LIN {X 771.523, Y -384.331, Z 83.55, A 0, B 90, C -0, E1 0, E2 0, E3 0, E4 0} C_DIS
LIN {X 767.677, Y -378.417, Z 83.55, A 0, B 90, C -0, E1 0, E2 0, E3 0, E4 0} C_DIS
LIN {X 766.611, Y -377.585, Z 83.55, A 0, B 90, C -0, E1 0, E2 0, E3 0, E4 0} C_DIS
LIN {X 765.394, Y -378.227, Z 83.55, A 0, B 90, C -0, E1 0, E2 0, E3 0, E4 0} C_DIS
LIN {X 760.024, Y -382.801, Z 83.55, A 0, B 90, C -0, E1 0, E2 0, E3 0, E4 0} C_DIS
LIN {X 758.756, Y -383.361, Z 83.55, A 0, B 90, C -0, E1 0, E2 0, E3 0, E4 0} C_DIS
LIN {X 757.411, Y -383.004, Z 83.55, A 0, B 90, C -0, E1 0, E2 0, E3 0, E4 0} C_DIS
LIN {X 751.124, Y -379.806, Z 83.55, A 0, B 90, C -0, E1 0, E2 0, E3 0, E4 0} C_DIS
LIN {X 749.785, Y -379.619, Z 83.55, A 0, B 90, C -0, E1 0, E2 0, E3 0, E4 0} C_DIS
LIN {X 749.052, Y -380.783, Z 83.55, A 0, B 90, C -0, E1 0, E2 0, E3 0, E4 0} C_DIS
LIN {X 746.688, Y -387.429, Z 83.55, A 0, B 90, C -0, E1 0, E2 0, E3 0, E4 0} C_DIS
LIN {X 745.87, Y -388.548, Z 83.55, A 0, B 90, C -0, E1 0, E2 0, E3 0, E4 0} C_DIS
LIN {X 744.527, Y -388.912, Z 83.55, A 0, B 90, C -0, E1 0, E2 0, E3 0, E4 0} C_DIS
LIN {X 737.483, Y -389.285, Z 83.55, A 0, B 90, C -0, E1 0, E2 0, E3 0, E4 0} C_DIS
LIN {X 736.23, Y -389.793, Z 83.55, A 0, B 90, C -0, E1 0, E2 0, E3 0, E4 0} C_DIS
LIN {X 736.177, Y -391.167, Z 83.55, A 0, B 90, C -0, E1 0, E2 0, E3 0, E4 0} C_DIS
LIN {X 737.453, Y -398.105, Z 83.55, A 0, B 90, C -0, E1 0, E2 0, E3 0, E4 0} C_DIS
LIN {X 737.304, Y -399.483, Z 83.55, A 0, B 90, C -0, E1 0, E2 0, E3 0, E4 0} C_DIS
LIN {X 736.323, Y -400.469, Z 83.55, A 0, B 90, C -0, E1 0, E2 0, E3 0, E4 0} C_DIS
LIN {X 730.41, Y -404.315, Z 83.55, A 0, B 90, C -0, E1 0, E2 0, E3 0, E4 0} C_DIS
LIN {X 729.578, Y -405.381, Z 83.55, A 0, B 90, C -0, E1 0, E2 0, E3 0, E4 0} C_DIS
LIN {X 730.22, Y -406.598, Z 83.55, A 0, B 90, C -0, E1 0, E2 0, E3 0, E4 0} C_DIS
LIN {X 734.793, Y -411.969, Z 83.55, A 0, B 90, C -0, E1 0, E2 0, E3 0, E4 0} C_DIS
LIN {X 735.354, Y -413.236, Z 83.55, A 0, B 90, C -0, E1 0, E2 0, E3 0, E4 0} C_DIS
LIN {X 734.997, Y -414.581, Z 83.55, A 0, B 90, C -0, E1 0, E2 0, E3 0, E4 0} C_DIS
LIN {X 731.798, Y -420.868, Z 83.55, A 0, B 90, C -0, E1 0, E2 0, E3 0, E4 0} C_DIS
LIN {X 731.611, Y -422.208, Z 83.55, A 0, B 90, C -0, E1 0, E2 0, E3 0, E4 0} C_DIS
LIN {X 732.775, Y -422.94, Z 83.55, A 0, B 90, C -0, E1 0, E2 0, E3 0, E4 0} C_DIS
LIN {X 739.421, Y -425.305, Z 83.55, A 0, B 90, C -0, E1 0, E2 0, E3 0, E4 0} C_DIS
LIN {X 740.541, Y -426.122, Z 83.55, A 0, B 90, C -0, E1 0, E2 0, E3 0, E4 0} C_DIS
LIN {X 740.904, Y -427.465, Z 83.55, A 0, B 90, C -0, E1 0, E2 0, E3 0, E4 0} C_DIS
LIN {X 741.278, Y -434.509, Z 83.55, A 0, B 90, C -0, E1 0, E2 0, E3 0, E4 0} C_DIS
LIN {X 741.785, Y -435.763, Z 83.55, A 0, B 90, C -0, E1 0, E2 0, E3 0, E4 0} C_DIS
LIN {X 743.16, Y -435.815, Z 83.55, A 0, B 90, C -0, E1 0, E2 0, E3 0, E4 0} C_DIS
LIN {X 750.098, Y -434.54, Z 83.55, A 0, B 90, C -0, E1 0, E2 0, E3 0, E4 0} C_DIS
LIN {X 751.476, Y -434.688, Z 83.55, A 0, B 90, C -0, E1 0, E2 0, E3 0, E4 0} C_DIS
LIN {X 752.462, Y -435.669, Z 83.55, A 0, B 90, C -0, E1 0, E2 0, E3 0, E4 0} C_DIS
LIN {X 756.308, Y -441.583, Z 83.55, A 0, B 90, C -0, E1 0, E2 0, E3 0, E4 0} C_DIS
LIN {X 757.374, Y -442.415, Z 83.55, A 0, B 90, C -0, E1 0, E2 0, E3 0, E4 0} C_DIS
LIN {X 758.591, Y -441.773, Z 83.55, A 0, B 90, C -0, E1 0, E2 0, E3 0, E4 0} C_DIS
LIN {X 763.961, Y -437.199, Z 83.55, A 0, B 90, C -0, E1 0, E2 0, E3 0, E4 0} C_DIS
LIN {X 765.229, Y -436.639, Z 83.55, A 0, B 90, C -0, E1 0, E2 0, E3 0, E4 0} C_DIS
LIN {X 766.573, Y -436.996, Z 83.55, A 0, B 90, C -0, E1 0, E2 0, E3 0, E4 0} C_DIS
LIN {X 772.861, Y -440.194, Z 83.55, A 0, B 90, C -0, E1 0, E2 0, E3 0, E4 0} C_DIS
LIN {X 774.2, Y -440.381, Z 83.55, A 0, B 90, C -0, E1 0, E2 0, E3 0, E4 0} C_DIS
LIN {X 774.933, Y -439.217, Z 83.55, A 0, B 90, C -0, E1 0, E2 0, E3 0, E4 0} C_DIS
LIN {X 777.297, Y -432.571, Z 83.55, A 0, B 90, C -0, E1 0, E2 0, E3 0, E4 0} C_DIS
LIN {X 778.115, Y -431.452, Z 83.55, A 0, B 90, C -0, E1 0, E2 0, E3 0, E4 0} C_DIS
LIN {X 779.458, Y -431.088, Z 83.55, A 0, B 90, C -0, E1 0, E2 0, E3 0, E4 0} C_DIS
LIN {X 786.502, Y -430.715, Z 83.55, A 0, B 90, C -0, E1 0, E2 0, E3 0, E4 0} C_DIS
LIN {X 787.755, Y -430.207, Z 83.55, A 0, B 90, C -0, E1 0, E2 0, E3 0, E4 0} C_DIS
LIN {X 787.808, Y -428.833, Z 83.55, A 0, B 90, C -0, E1 0, E2 0, E3 0, E4 0} C_DIS
LIN {X 786.532, Y -421.895, Z 83.55, A 0, B 90, C -0, E1 0, E2 0, E3 0, E4 0} C_DIS
LIN {X 786.681, Y -420.517, Z 83.55, A 0, B 90, C -0, E1 0, E2 0, E3 0, E4 0} C_DIS
LIN {X 787.662, Y -419.531, Z 83.55, A 0, B 90, C -0, E1 0, E2 0, E3 0, E4 0} C_DIS
LIN {X 793.575, Y -415.685, Z 83.55, A 0, B 90, C -0, E1 0, E2 0, E3 0, E4 0} C_DIS
LIN {X 794.407, Y -414.619, Z 83.55, A 0, B 90, C -0, E1 0, E2 0, E3 0, E4 0} C_DIS
LIN {X 793.765, Y -413.402, Z 83.55, A 0, B 90, C -0, E1 0, E2 0, E3 0, E4 0} C_DIS
LIN {X 789.192, Y -408.031, Z 83.55, A 0, B 90, C -0, E1 0, E2 0, E3 0, E4 0} C_DIS
LIN {X 788.631, Y -406.764, Z 83.55, A 0, B 90, C -0, E1 0, E2 0, E3 0, E4 0} C_DIS
LIN {X 788.988, Y -405.419, Z 83.55, A 0, B 90, C -0, E1 0, E2 0, E3 0, E4 0} C_DIS
LIN {X 792.186, Y -399.132, Z 83.55, A 0, B 90, C -0, E1 0, E2 0, E3 0, E4 0} C_DIS
LIN {X 792.374, Y -397.792, Z 83.55, A 0, B 90, C -0, E1 0, E2 0, E3 0, E4 0} C_DIS
LIN {X 791.209, Y -397.06, Z 83.55, A 0, B 90, C -0, E1 0, E2 0, E3 0, E4 0} C_DIS
LIN {X 784.564, Y -394.695, Z 83.55, A 0, B 90, C -0, E1 0, E2 0, E3 0, E4 0} C_DIS
LIN {X 783.444, Y -393.878, Z 83.55, A 0, B 90, C -0, E1 0, E2 0, E3 0, E4 0} C_DIS
LIN {X 783.081, Y -392.535, Z 83.55, A 0, B 90, C -0, E1 0, E2 0, E3 0, E4 0} C_DIS
LIN {X 782.707, Y -385.491, Z 83.55, A 0, B 90, C -0, E1 0, E2 0, E3 0, E4 0} C_DIS
LIN {X 782.2, Y -384.237, Z 83.55, A 0, B 90, C -0, E1 0, E2 0, E3 0, E4 0} C_DIS
LIN {X 780.825, Y -384.185, Z 83.55, A 0, B 90, C -0, E1 0, E2 0, E3 0, E4 0} C_DIS
LIN {X 775.275, Y -385.205, Z 83.55, A 0, B 90, C -0, E1 0, E2 0, E3 0, E4 0} C_DIS
LIN {X 773.608, Y -385.498, Z 84.2, A 0, B 90, C -0, E1 0, E2 0, E3 0, E4 0} C_DIS
LIN {X 772.237, Y -385.362, Z 84.2, A 0, B 90, C -0, E1 0, E2 0, E3 0, E4 0} C_DIS
LIN {X 771.248, Y -384.395, Z 84.2, A 0, B 90, C -0, E1 0, E2 0, E3 0, E4 0} C_DIS
LIN {X 767.373, Y -378.549, Z 84.2, A 0, B 90, C -0, E1 0, E2 0, E3 0, E4 0} C_DIS
LIN {X 766.306, Y -377.731, Z 84.2, A 0, B 90, C -0, E1 0, E2 0, E3 0, E4 0} C_DIS
LIN {X 765.101, Y -378.379, Z 84.2, A 0, B 90, C -0, E1 0, E2 0, E3 0, E4 0} C_DIS
LIN {X 759.801, Y -382.973, Z 84.2, A 0, B 90, C -0, E1 0, E2 0, E3 0, E4 0} C_DIS
LIN {X 758.545, Y -383.541, Z 84.2, A 0, B 90, C -0, E1 0, E2 0, E3 0, E4 0} C_DIS
LIN {X 757.205, Y -383.198, Z 84.2, A 0, B 90, C -0, E1 0, E2 0, E3 0, E4 0} C_DIS
LIN {X 750.926, Y -380.072, Z 84.2, A 0, B 90, C -0, E1 0, E2 0, E3 0, E4 0} C_DIS
LIN {X 749.593, Y -379.897, Z 84.2, A 0, B 90, C -0, E1 0, E2 0, E3 0, E4 0} C_DIS
LIN {X 748.875, Y -381.061, Z 84.2, A 0, B 90, C -0, E1 0, E2 0, E3 0, E4 0} C_DIS
LIN {X 746.581, Y -387.69, Z 84.2, A 0, B 90, C -0, E1 0, E2 0, E3 0, E4 0} C_DIS
LIN {X 745.778, Y -388.81, Z 84.2, A 0, B 90, C -0, E1 0, E2 0, E3 0, E4 0} C_DIS
LIN {X 744.446, Y -389.182, Z 84.2, A 0, B 90, C -0, E1 0, E2 0, E3 0, E4 0} C_DIS
LIN {X 737.445, Y -389.615, Z 84.2, A 0, B 90, C -0, E1 0, E2 0, E3 0, E4 0} C_DIS
LIN {X 736.203, Y -390.13, Z 84.2, A 0, B 90, C -0, E1 0, E2 0, E3 0, E4 0} C_DIS
LIN {X 736.163, Y -391.497, Z 84.2, A 0, B 90, C -0, E1 0, E2 0, E3 0, E4 0} C_DIS
LIN {X 737.491, Y -398.384, Z 84.2, A 0, B 90, C -0, E1 0, E2 0, E3 0, E4 0} C_DIS
LIN {X 737.355, Y -399.756, Z 84.2, A 0, B 90, C -0, E1 0, E2 0, E3 0, E4 0} C_DIS
LIN {X 736.388, Y -400.745, Z 84.2, A 0, B 90, C -0, E1 0, E2 0, E3 0, E4 0} C_DIS
LIN {X 730.541, Y -404.619, Z 84.2, A 0, B 90, C -0, E1 0, E2 0, E3 0, E4 0} C_DIS
LIN {X 729.723, Y -405.687, Z 84.2, A 0, B 90, C -0, E1 0, E2 0, E3 0, E4 0} C_DIS
LIN {X 730.372, Y -406.891, Z 84.2, A 0, B 90, C -0, E1 0, E2 0, E3 0, E4 0} C_DIS
LIN {X 734.965, Y -412.191, Z 84.2, A 0, B 90, C -0, E1 0, E2 0, E3 0, E4 0} C_DIS
LIN {X 735.534, Y -413.447, Z 84.2, A 0, B 90, C -0, E1 0, E2 0, E3 0, E4 0} C_DIS
LIN {X 735.19, Y -414.787, Z 84.2, A 0, B 90, C -0, E1 0, E2 0, E3 0, E4 0} C_DIS
LIN {X 732.064, Y -421.066, Z 84.2, A 0, B 90, C -0, E1 0, E2 0, E3 0, E4 0} C_DIS
LIN {X 731.89, Y -422.399, Z 84.2, A 0, B 90, C -0, E1 0, E2 0, E3 0, E4 0} C_DIS
LIN {X 733.054, Y -423.118, Z 84.2, A 0, B 90, C -0, E1 0, E2 0, E3 0, E4 0} C_DIS
LIN {X 739.682, Y -425.411, Z 84.2, A 0, B 90, C -0, E1 0, E2 0, E3 0, E4 0} C_DIS
LIN {X 740.802, Y -426.215, Z 84.2, A 0, B 90, C -0, E1 0, E2 0, E3 0, E4 0} C_DIS
LIN {X 741.175, Y -427.547, Z 84.2, A 0, B 90, C -0, E1 0, E2 0, E3 0, E4 0} C_DIS
LIN {X 741.607, Y -434.547, Z 84.2, A 0, B 90, C -0, E1 0, E2 0, E3 0, E4 0} C_DIS
LIN {X 742.122, Y -435.79, Z 84.2, A 0, B 90, C -0, E1 0, E2 0, E3 0, E4 0} C_DIS
LIN {X 743.49, Y -435.83, Z 84.2, A 0, B 90, C -0, E1 0, E2 0, E3 0, E4 0} C_DIS
LIN {X 750.377, Y -434.502, Z 84.2, A 0, B 90, C -0, E1 0, E2 0, E3 0, E4 0} C_DIS
LIN {X 751.748, Y -434.638, Z 84.2, A 0, B 90, C -0, E1 0, E2 0, E3 0, E4 0} C_DIS
LIN {X 752.737, Y -435.605, Z 84.2, A 0, B 90, C -0, E1 0, E2 0, E3 0, E4 0} C_DIS
LIN {X 756.612, Y -441.451, Z 84.2, A 0, B 90, C -0, E1 0, E2 0, E3 0, E4 0} C_DIS
LIN {X 757.679, Y -442.269, Z 84.2, A 0, B 90, C -0, E1 0, E2 0, E3 0, E4 0} C_DIS
LIN {X 758.884, Y -441.621, Z 84.2, A 0, B 90, C -0, E1 0, E2 0, E3 0, E4 0} C_DIS
LIN {X 764.184, Y -437.027, Z 84.2, A 0, B 90, C -0, E1 0, E2 0, E3 0, E4 0} C_DIS
LIN {X 765.44, Y -436.459, Z 84.2, A 0, B 90, C -0, E1 0, E2 0, E3 0, E4 0} C_DIS
LIN {X 766.78, Y -436.802, Z 84.2, A 0, B 90, C -0, E1 0, E2 0, E3 0, E4 0} C_DIS
LIN {X 773.058, Y -439.928, Z 84.2, A 0, B 90, C -0, E1 0, E2 0, E3 0, E4 0} C_DIS
LIN {X 774.392, Y -440.103, Z 84.2, A 0, B 90, C -0, E1 0, E2 0, E3 0, E4 0} C_DIS
LIN {X 775.11, Y -438.939, Z 84.2, A 0, B 90, C -0, E1 0, E2 0, E3 0, E4 0} C_DIS
LIN {X 777.404, Y -432.31, Z 84.2, A 0, B 90, C -0, E1 0, E2 0, E3 0, E4 0} C_DIS
LIN {X 778.207, Y -431.19, Z 84.2, A 0, B 90, C -0, E1 0, E2 0, E3 0, E4 0} C_DIS
LIN {X 779.539, Y -430.818, Z 84.2, A 0, B 90, C -0, E1 0, E2 0, E3 0, E4 0} C_DIS
LIN {X 786.54, Y -430.385, Z 84.2, A 0, B 90, C -0, E1 0, E2 0, E3 0, E4 0} C_DIS
LIN {X 787.782, Y -429.87, Z 84.2, A 0, B 90, C -0, E1 0, E2 0, E3 0, E4 0} C_DIS
LIN {X 787.822, Y -428.503, Z 84.2, A 0, B 90, C -0, E1 0, E2 0, E3 0, E4 0} C_DIS
LIN {X 786.494, Y -421.616, Z 84.2, A 0, B 90, C -0, E1 0, E2 0, E3 0, E4 0} C_DIS
LIN {X 786.63, Y -420.244, Z 84.2, A 0, B 90, C -0, E1 0, E2 0, E3 0, E4 0} C_DIS
LIN {X 787.597, Y -419.255, Z 84.2, A 0, B 90, C -0, E1 0, E2 0, E3 0, E4 0} C_DIS
LIN {X 793.444, Y -415.381, Z 84.2, A 0, B 90, C -0, E1 0, E2 0, E3 0, E4 0} C_DIS
LIN {X 794.262, Y -414.313, Z 84.2, A 0, B 90, C -0, E1 0, E2 0, E3 0, E4 0} C_DIS
LIN {X 793.613, Y -413.109, Z 84.2, A 0, B 90, C -0, E1 0, E2 0, E3 0, E4 0} C_DIS
LIN {X 789.02, Y -407.809, Z 84.2, A 0, B 90, C -0, E1 0, E2 0, E3 0, E4 0} C_DIS
LIN {X 788.451, Y -406.553, Z 84.2, A 0, B 90, C -0, E1 0, E2 0, E3 0, E4 0} C_DIS
LIN {X 788.795, Y -405.213, Z 84.2, A 0, B 90, C -0, E1 0, E2 0, E3 0, E4 0} C_DIS
LIN {X 791.92, Y -398.934, Z 84.2, A 0, B 90, C -0, E1 0, E2 0, E3 0, E4 0} C_DIS
LIN {X 792.095, Y -397.601, Z 84.2, A 0, B 90, C -0, E1 0, E2 0, E3 0, E4 0} C_DIS
LIN {X 790.931, Y -396.882, Z 84.2, A 0, B 90, C -0, E1 0, E2 0, E3 0, E4 0} C_DIS
LIN {X 784.303, Y -394.589, Z 84.2, A 0, B 90, C -0, E1 0, E2 0, E3 0, E4 0} C_DIS
LIN {X 783.183, Y -393.785, Z 84.2, A 0, B 90, C -0, E1 0, E2 0, E3 0, E4 0} C_DIS
LIN {X 782.81, Y -392.453, Z 84.2, A 0, B 90, C -0, E1 0, E2 0, E3 0, E4 0} C_DIS
LIN {X 782.378, Y -385.453, Z 84.2, A 0, B 90, C -0, E1 0, E2 0, E3 0, E4 0} C_DIS
LIN {X 781.862, Y -384.21, Z 84.2, A 0, B 90, C -0, E1 0, E2 0, E3 0, E4 0} C_DIS
LIN {X 780.495, Y -384.17, Z 84.2, A 0, B 90, C -0, E1 0, E2 0, E3 0, E4 0} C_DIS
LIN {X 774.986, Y -385.233, Z 84.2, A 0, B 90, C -0, E1 0, E2 0, E3 0, E4 0} C_DIS
LIN {X 773.332, Y -385.538, Z 84.85, A 0, B 90, C -0, E1 0, E2 0, E3 0, E4 0} C_DIS
LIN {X 771.966, Y -385.414, Z 84.85, A 0, B 90, C -0, E1 0, E2 0, E3 0, E4 0} C_DIS
LIN {X 770.975, Y -384.461, Z 84.85, A 0, B 90, C -0, E1 0, E2 0, E3 0, E4 0} C_DIS
LIN {X 767.072, Y -378.681, Z 84.85, A 0, B 90, C -0, E1 0, E2 0, E3 0, E4 0} C_DIS
LIN {X 766.004, Y -377.877, Z 84.85, A 0, B 90, C -0, E1 0, E2 0, E3 0, E4 0} C_DIS
LIN {X 764.812, Y -378.533, Z 84.85, A 0, B 90, C -0, E1 0, E2 0, E3 0, E4 0} C_DIS
LIN {X 759.581, Y -383.145, Z 84.85, A 0, B 90, C -0, E1 0, E2 0, E3 0, E4 0} C_DIS
LIN {X 758.337, Y -383.721, Z 84.85, A 0, B 90, C -0, E1 0, E2 0, E3 0, E4 0} C_DIS
LIN {X 757.002, Y -383.392, Z 84.85, A 0, B 90, C -0, E1 0, E2 0, E3 0, E4 0} C_DIS
LIN {X 750.732, Y -380.337, Z 84.85, A 0, B 90, C -0, E1 0, E2 0, E3 0, E4 0} C_DIS
LIN {X 749.405, Y -380.175, Z 84.85, A 0, B 90, C -0, E1 0, E2 0, E3 0, E4 0} C_DIS
LIN {X 748.701, Y -381.339, Z 84.85, A 0, B 90, C -0, E1 0, E2 0, E3 0, E4 0} C_DIS
LIN {X 746.477, Y -387.949, Z 84.85, A 0, B 90, C -0, E1 0, E2 0, E3 0, E4 0} C_DIS
LIN {X 745.688, Y -389.069, Z 84.85, A 0, B 90, C -0, E1 0, E2 0, E3 0, E4 0} C_DIS
LIN {X 744.367, Y -389.452, Z 84.85, A 0, B 90, C -0, E1 0, E2 0, E3 0, E4 0} C_DIS
LIN {X 737.409, Y -389.942, Z 84.85, A 0, B 90, C -0, E1 0, E2 0, E3 0, E4 0} C_DIS
LIN {X 736.179, Y -390.465, Z 84.85, A 0, B 90, C -0, E1 0, E2 0, E3 0, E4 0} C_DIS
LIN {X 736.151, Y -391.824, Z 84.85, A 0, B 90, C -0, E1 0, E2 0, E3 0, E4 0} C_DIS
LIN {X 737.53, Y -398.661, Z 84.85, A 0, B 90, C -0, E1 0, E2 0, E3 0, E4 0} C_DIS
LIN {X 737.407, Y -400.026, Z 84.85, A 0, B 90, C -0, E1 0, E2 0, E3 0, E4 0} C_DIS
LIN {X 736.454, Y -401.017, Z 84.85, A 0, B 90, C -0, E1 0, E2 0, E3 0, E4 0} C_DIS
LIN {X 730.674, Y -404.92, Z 84.85, A 0, B 90, C -0, E1 0, E2 0, E3 0, E4 0} C_DIS
LIN {X 729.87, Y -405.989, Z 84.85, A 0, B 90, C -0, E1 0, E2 0, E3 0, E4 0} C_DIS
LIN {X 730.525, Y -407.181, Z 84.85, A 0, B 90, C -0, E1 0, E2 0, E3 0, E4 0} C_DIS
LIN {X 735.138, Y -412.411, Z 84.85, A 0, B 90, C -0, E1 0, E2 0, E3 0, E4 0} C_DIS
LIN {X 735.714, Y -413.655, Z 84.85, A 0, B 90, C -0, E1 0, E2 0, E3 0, E4 0} C_DIS
LIN {X 735.384, Y -414.99, Z 84.85, A 0, B 90, C -0, E1 0, E2 0, E3 0, E4 0} C_DIS
LIN {X 732.33, Y -421.26, Z 84.85, A 0, B 90, C -0, E1 0, E2 0, E3 0, E4 0} C_DIS
LIN {X 732.168, Y -422.588, Z 84.85, A 0, B 90, C -0, E1 0, E2 0, E3 0, E4 0} C_DIS
LIN {X 733.331, Y -423.292, Z 84.85, A 0, B 90, C -0, E1 0, E2 0, E3 0, E4 0} C_DIS
LIN {X 739.941, Y -425.515, Z 84.85, A 0, B 90, C -0, E1 0, E2 0, E3 0, E4 0} C_DIS
LIN {X 741.062, Y -426.305, Z 84.85, A 0, B 90, C -0, E1 0, E2 0, E3 0, E4 0} C_DIS
LIN {X 741.444, Y -427.626, Z 84.85, A 0, B 90, C -0, E1 0, E2 0, E3 0, E4 0} C_DIS
LIN {X 741.934, Y -434.583, Z 84.85, A 0, B 90, C -0, E1 0, E2 0, E3 0, E4 0} C_DIS
LIN {X 742.457, Y -435.814, Z 84.85, A 0, B 90, C -0, E1 0, E2 0, E3 0, E4 0} C_DIS
LIN {X 743.817, Y -435.842, Z 84.85, A 0, B 90, C -0, E1 0, E2 0, E3 0, E4 0} C_DIS
LIN {X 750.653, Y -434.462, Z 84.85, A 0, B 90, C -0, E1 0, E2 0, E3 0, E4 0} C_DIS
LIN {X 752.018, Y -434.586, Z 84.85, A 0, B 90, C -0, E1 0, E2 0, E3 0, E4 0} C_DIS
LIN {X 753.01, Y -435.539, Z 84.85, A 0, B 90, C -0, E1 0, E2 0, E3 0, E4 0} C_DIS
LIN {X 756.913, Y -441.319, Z 84.85, A 0, B 90, C -0, E1 0, E2 0, E3 0, E4 0} C_DIS
LIN {X 757.981, Y -442.123, Z 84.85, A 0, B 90, C -0, E1 0, E2 0, E3 0, E4 0} C_DIS
LIN {X 759.173, Y -441.467, Z 84.85, A 0, B 90, C -0, E1 0, E2 0, E3 0, E4 0} C_DIS
LIN {X 764.404, Y -436.855, Z 84.85, A 0, B 90, C -0, E1 0, E2 0, E3 0, E4 0} C_DIS
LIN {X 765.648, Y -436.279, Z 84.85, A 0, B 90, C -0, E1 0, E2 0, E3 0, E4 0} C_DIS
LIN {X 766.983, Y -436.608, Z 84.85, A 0, B 90, C -0, E1 0, E2 0, E3 0, E4 0} C_DIS
LIN {X 773.253, Y -439.663, Z 84.85, A 0, B 90, C -0, E1 0, E2 0, E3 0, E4 0} C_DIS
LIN {X 774.58, Y -439.825, Z 84.85, A 0, B 90, C -0, E1 0, E2 0, E3 0, E4 0} C_DIS
LIN {X 775.284, Y -438.661, Z 84.85, A 0, B 90, C -0, E1 0, E2 0, E3 0, E4 0} C_DIS
LIN {X 777.508, Y -432.051, Z 84.85, A 0, B 90, C -0, E1 0, E2 0, E3 0, E4 0} C_DIS
LIN {X 778.297, Y -430.931, Z 84.85, A 0, B 90, C -0, E1 0, E2 0, E3 0, E4 0} C_DIS
LIN {X 779.618, Y -430.548, Z 84.85, A 0, B 90, C -0, E1 0, E2 0, E3 0, E4 0} C_DIS
LIN {X 786.576, Y -430.058, Z 84.85, A 0, B 90, C -0, E1 0, E2 0, E3 0, E4 0} C_DIS
LIN {X 787.806, Y -429.535, Z 84.85, A 0, B 90, C -0, E1 0, E2 0, E3 0, E4 0} C_DIS
LIN {X 787.834, Y -428.176, Z 84.85, A 0, B 90, C -0, E1 0, E2 0, E3 0, E4 0} C_DIS
LIN {X 786.455, Y -421.339, Z 84.85, A 0, B 90, C -0, E1 0, E2 0, E3 0, E4 0} C_DIS
LIN {X 786.578, Y -419.974, Z 84.85, A 0, B 90, C -0, E1 0, E2 0, E3 0, E4 0} C_DIS
LIN {X 787.531, Y -418.983, Z 84.85, A 0, B 90, C -0, E1 0, E2 0, E3 0, E4 0} C_DIS
LIN {X 793.311, Y -415.08, Z 84.85, A 0, B 90, C -0, E1 0, E2 0, E3 0, E4 0} C_DIS
LIN {X 794.115, Y -414.011, Z 84.85, A 0, B 90, C -0, E1 0, E2 0, E3 0, E4 0} C_DIS
LIN {X 793.46, Y -412.819, Z 84.85, A 0, B 90, C -0, E1 0, E2 0, E3 0, E4 0} C_DIS
LIN {X 788.847, Y -407.589, Z 84.85, A 0, B 90, C -0, E1 0, E2 0, E3 0, E4 0} C_DIS
LIN {X 788.271, Y -406.345, Z 84.85, A 0, B 90, C -0, E1 0, E2 0, E3 0, E4 0} C_DIS
LIN {X 788.601, Y -405.01, Z 84.85, A 0, B 90, C -0, E1 0, E2 0, E3 0, E4 0} C_DIS
LIN {X 791.655, Y -398.74, Z 84.85, A 0, B 90, C -0, E1 0, E2 0, E3 0, E4 0} C_DIS
LIN {X 791.817, Y -397.412, Z 84.85, A 0, B 90, C -0, E1 0, E2 0, E3 0, E4 0} C_DIS
LIN {X 790.654, Y -396.708, Z 84.85, A 0, B 90, C -0, E1 0, E2 0, E3 0, E4 0} C_DIS
LIN {X 784.044, Y -394.485, Z 84.85, A 0, B 90, C -0, E1 0, E2 0, E3 0, E4 0} C_DIS
LIN {X 782.923, Y -393.695, Z 84.85, A 0, B 90, C -0, E1 0, E2 0, E3 0, E4 0} C_DIS
LIN {X 782.541, Y -392.374, Z 84.85, A 0, B 90, C -0, E1 0, E2 0, E3 0, E4 0} C_DIS
LIN {X 782.051, Y -385.417, Z 84.85, A 0, B 90, C -0, E1 0, E2 0, E3 0, E4 0} C_DIS
LIN {X 781.528, Y -384.186, Z 84.85, A 0, B 90, C -0, E1 0, E2 0, E3 0, E4 0} C_DIS
LIN {X 780.168, Y -384.158, Z 84.85, A 0, B 90, C -0, E1 0, E2 0, E3 0, E4 0} C_DIS
LIN {X 774.699, Y -385.262, Z 84.85, A 0, B 90, C -0, E1 0, E2 0, E3 0, E4 0} C_DIS
LIN {X 773.057, Y -385.579, Z 85.5, A 0, B 90, C -0, E1 0, E2 0, E3 0, E4 0} C_DIS
LIN {X 771.699, Y -385.468, Z 85.5, A 0, B 90, C -0, E1 0, E2 0, E3 0, E4 0} C_DIS
LIN {X 770.705, Y -384.529, Z 85.5, A 0, B 90, C -0, E1 0, E2 0, E3 0, E4 0} C_DIS
LIN {X 766.775, Y -378.815, Z 85.5, A 0, B 90, C -0, E1 0, E2 0, E3 0, E4 0} C_DIS
LIN {X 765.706, Y -378.025, Z 85.5, A 0, B 90, C -0, E1 0, E2 0, E3 0, E4 0} C_DIS
LIN {X 764.526, Y -378.686, Z 85.5, A 0, B 90, C -0, E1 0, E2 0, E3 0, E4 0} C_DIS
LIN {X 759.364, Y -383.318, Z 85.5, A 0, B 90, C -0, E1 0, E2 0, E3 0, E4 0} C_DIS
LIN {X 758.133, Y -383.901, Z 85.5, A 0, B 90, C -0, E1 0, E2 0, E3 0, E4 0} C_DIS
LIN {X 756.802, Y -383.585, Z 85.5, A 0, B 90, C -0, E1 0, E2 0, E3 0, E4 0} C_DIS
LIN {X 750.541, Y -380.602, Z 85.5, A 0, B 90, C -0, E1 0, E2 0, E3 0, E4 0} C_DIS
LIN {X 749.22, Y -380.452, Z 85.5, A 0, B 90, C -0, E1 0, E2 0, E3 0, E4 0} C_DIS
LIN {X 748.53, Y -381.615, Z 85.5, A 0, B 90, C -0, E1 0, E2 0, E3 0, E4 0} C_DIS
LIN {X 746.376, Y -388.207, Z 85.5, A 0, B 90, C -0, E1 0, E2 0, E3 0, E4 0} C_DIS
LIN {X 745.6, Y -389.328, Z 85.5, A 0, B 90, C -0, E1 0, E2 0, E3 0, E4 0} C_DIS
LIN {X 744.29, Y -389.719, Z 85.5, A 0, B 90, C -0, E1 0, E2 0, E3 0, E4 0} C_DIS
LIN {X 737.377, Y -390.266, Z 85.5, A 0, B 90, C -0, E1 0, E2 0, E3 0, E4 0} C_DIS
LIN {X 736.157, Y -390.797, Z 85.5, A 0, B 90, C -0, E1 0, E2 0, E3 0, E4 0} C_DIS
LIN {X 736.141, Y -392.149, Z 85.5, A 0, B 90, C -0, E1 0, E2 0, E3 0, E4 0} C_DIS
LIN {X 737.571, Y -398.935, Z 85.5, A 0, B 90, C -0, E1 0, E2 0, E3 0, E4 0} C_DIS
LIN {X 737.46, Y -400.293, Z 85.5, A 0, B 90, C -0, E1 0, E2 0, E3 0, E4 0} C_DIS
LIN {X 736.521, Y -401.287, Z 85.5, A 0, B 90, C -0, E1 0, E2 0, E3 0, E4 0} C_DIS
LIN {X 730.807, Y -405.218, Z 85.5, A 0, B 90, C -0, E1 0, E2 0, E3 0, E4 0} C_DIS
LIN {X 730.017, Y -406.287, Z 85.5, A 0, B 90, C -0, E1 0, E2 0, E3 0, E4 0} C_DIS
LIN {X 730.679, Y -407.466, Z 85.5, A 0, B 90, C -0, E1 0, E2 0, E3 0, E4 0} C_DIS
LIN {X 735.311, Y -412.628, Z 85.5, A 0, B 90, C -0, E1 0, E2 0, E3 0, E4 0} C_DIS
LIN {X 735.894, Y -413.86, Z 85.5, A 0, B 90, C -0, E1 0, E2 0, E3 0, E4 0} C_DIS
LIN {X 735.577, Y -415.19, Z 85.5, A 0, B 90, C -0, E1 0, E2 0, E3 0, E4 0} C_DIS
LIN {X 732.594, Y -421.451, Z 85.5, A 0, B 90, C -0, E1 0, E2 0, E3 0, E4 0} C_DIS
LIN {X 732.444, Y -422.772, Z 85.5, A 0, B 90, C -0, E1 0, E2 0, E3 0, E4 0} C_DIS
LIN {X 733.607, Y -423.463, Z 85.5, A 0, B 90, C -0, E1 0, E2 0, E3 0, E4 0} C_DIS
LIN {X 740.199, Y -425.617, Z 85.5, A 0, B 90, C -0, E1 0, E2 0, E3 0, E4 0} C_DIS
LIN {X 741.32, Y -426.392, Z 85.5, A 0, B 90, C -0, E1 0, E2 0, E3 0, E4 0} C_DIS
LIN {X 741.712, Y -427.702, Z 85.5, A 0, B 90, C -0, E1 0, E2 0, E3 0, E4 0} C_DIS
LIN {X 742.258, Y -434.616, Z 85.5, A 0, B 90, C -0, E1 0, E2 0, E3 0, E4 0} C_DIS
LIN {X 742.789, Y -435.835, Z 85.5, A 0, B 90, C -0, E1 0, E2 0, E3 0, E4 0} C_DIS
LIN {X 744.142, Y -435.852, Z 85.5, A 0, B 90, C -0, E1 0, E2 0, E3 0, E4 0} C_DIS
LIN {X 750.927, Y -434.421, Z 85.5, A 0, B 90, C -0, E1 0, E2 0, E3 0, E4 0} C_DIS
LIN {X 752.286, Y -434.532, Z 85.5, A 0, B 90, C -0, E1 0, E2 0, E3 0, E4 0} C_DIS
LIN {X 753.28, Y -435.471, Z 85.5, A 0, B 90, C -0, E1 0, E2 0, E3 0, E4 0} C_DIS
LIN {X 757.21, Y -441.185, Z 85.5, A 0, B 90, C -0, E1 0, E2 0, E3 0, E4 0} C_DIS
LIN {X 758.279, Y -441.975, Z 85.5, A 0, B 90, C -0, E1 0, E2 0, E3 0, E4 0} C_DIS
LIN {X 759.459, Y -441.314, Z 85.5, A 0, B 90, C -0, E1 0, E2 0, E3 0, E4 0} C_DIS
LIN {X 764.62, Y -436.682, Z 85.5, A 0, B 90, C -0, E1 0, E2 0, E3 0, E4 0} C_DIS
LIN {X 765.852, Y -436.099, Z 85.5, A 0, B 90, C -0, E1 0, E2 0, E3 0, E4 0} C_DIS
LIN {X 767.183, Y -436.415, Z 85.5, A 0, B 90, C -0, E1 0, E2 0, E3 0, E4 0} C_DIS
LIN {X 773.443, Y -439.398, Z 85.5, A 0, B 90, C -0, E1 0, E2 0, E3 0, E4 0} C_DIS
LIN {X 774.765, Y -439.548, Z 85.5, A 0, B 90, C -0, E1 0, E2 0, E3 0, E4 0} C_DIS
LIN {X 775.455, Y -438.385, Z 85.5, A 0, B 90, C -0, E1 0, E2 0, E3 0, E4 0} C_DIS
LIN {X 777.609, Y -431.793, Z 85.5, A 0, B 90, C -0, E1 0, E2 0, E3 0, E4 0} C_DIS
LIN {X 778.385, Y -430.672, Z 85.5, A 0, B 90, C -0, E1 0, E2 0, E3 0, E4 0} C_DIS
LIN {X 779.695, Y -430.281, Z 85.5, A 0, B 90, C -0, E1 0, E2 0, E3 0, E4 0} C_DIS
LIN {X 786.608, Y -429.734, Z 85.5, A 0, B 90, C -0, E1 0, E2 0, E3 0, E4 0} C_DIS
LIN {X 787.828, Y -429.203, Z 85.5, A 0, B 90, C -0, E1 0, E2 0, E3 0, E4 0} C_DIS
LIN {X 787.844, Y -427.851, Z 85.5, A 0, B 90, C -0, E1 0, E2 0, E3 0, E4 0} C_DIS
LIN {X 786.414, Y -421.065, Z 85.5, A 0, B 90, C -0, E1 0, E2 0, E3 0, E4 0} C_DIS
LIN {X 786.524, Y -419.707, Z 85.5, A 0, B 90, C -0, E1 0, E2 0, E3 0, E4 0} C_DIS
LIN {X 787.464, Y -418.713, Z 85.5, A 0, B 90, C -0, E1 0, E2 0, E3 0, E4 0} C_DIS
LIN {X 793.177, Y -414.782, Z 85.5, A 0, B 90, C -0, E1 0, E2 0, E3 0, E4 0} C_DIS
LIN {X 793.968, Y -413.713, Z 85.5, A 0, B 90, C -0, E1 0, E2 0, E3 0, E4 0} C_DIS
LIN {X 793.306, Y -412.534, Z 85.5, A 0, B 90, C -0, E1 0, E2 0, E3 0, E4 0} C_DIS
LIN {X 788.674, Y -407.372, Z 85.5, A 0, B 90, C -0, E1 0, E2 0, E3 0, E4 0} C_DIS
LIN {X 788.091, Y -406.14, Z 85.5, A 0, B 90, C -0, E1 0, E2 0, E3 0, E4 0} C_DIS
LIN {X 788.407, Y -404.81, Z 85.5, A 0, B 90, C -0, E1 0, E2 0, E3 0, E4 0} C_DIS
LIN {X 791.391, Y -398.549, Z 85.5, A 0, B 90, C -0, E1 0, E2 0, E3 0, E4 0} C_DIS
LIN {X 791.541, Y -397.228, Z 85.5, A 0, B 90, C -0, E1 0, E2 0, E3 0, E4 0} C_DIS
LIN {X 790.378, Y -396.537, Z 85.5, A 0, B 90, C -0, E1 0, E2 0, E3 0, E4 0} C_DIS
LIN {X 783.786, Y -394.383, Z 85.5, A 0, B 90, C -0, E1 0, E2 0, E3 0, E4 0} C_DIS
LIN {X 782.665, Y -393.608, Z 85.5, A 0, B 90, C -0, E1 0, E2 0, E3 0, E4 0} C_DIS
LIN {X 782.273, Y -392.298, Z 85.5, A 0, B 90, C -0, E1 0, E2 0, E3 0, E4 0} C_DIS
LIN {X 781.727, Y -385.384, Z 85.5, A 0, B 90, C -0, E1 0, E2 0, E3 0, E4 0} C_DIS
LIN {X 781.196, Y -384.165, Z 85.5, A 0, B 90, C -0, E1 0, E2 0, E3 0, E4 0} C_DIS
LIN {X 779.843, Y -384.148, Z 85.5, A 0, B 90, C -0, E1 0, E2 0, E3 0, E4 0} C_DIS
LIN {X 774.415, Y -385.293, Z 85.5, A 0, B 90, C -0, E1 0, E2 0, E3 0, E4 0} C_DIS
LIN {X 772.786, Y -385.622, Z 86.15, A 0, B 90, C -0, E1 0, E2 0, E3 0, E4 0} C_DIS
LIN {X 771.434, Y -385.523, Z 86.15, A 0, B 90, C -0, E1 0, E2 0, E3 0, E4 0} C_DIS
LIN {X 770.438, Y -384.598, Z 86.15, A 0, B 90, C -0, E1 0, E2 0, E3 0, E4 0} C_DIS
LIN {X 766.481, Y -378.95, Z 86.15, A 0, B 90, C -0, E1 0, E2 0, E3 0, E4 0} C_DIS
LIN {X 765.411, Y -378.173, Z 86.15, A 0, B 90, C -0, E1 0, E2 0, E3 0, E4 0} C_DIS
LIN {X 764.244, Y -378.841, Z 86.15, A 0, B 90, C -0, E1 0, E2 0, E3 0, E4 0} C_DIS
LIN {X 759.151, Y -383.491, Z 86.15, A 0, B 90, C -0, E1 0, E2 0, E3 0, E4 0} C_DIS
LIN {X 757.931, Y -384.081, Z 86.15, A 0, B 90, C -0, E1 0, E2 0, E3 0, E4 0} C_DIS
LIN {X 756.605, Y -383.778, Z 86.15, A 0, B 90, C -0, E1 0, E2 0, E3 0, E4 0} C_DIS
LIN {X 750.354, Y -380.865, Z 86.15, A 0, B 90, C -0, E1 0, E2 0, E3 0, E4 0} C_DIS
LIN {X 749.039, Y -380.728, Z 86.15, A 0, B 90, C -0, E1 0, E2 0, E3 0, E4 0} C_DIS
LIN {X 748.363, Y -381.89, Z 86.15, A 0, B 90, C -0, E1 0, E2 0, E3 0, E4 0} C_DIS
LIN {X 746.277, Y -388.463, Z 86.15, A 0, B 90, C -0, E1 0, E2 0, E3 0, E4 0} C_DIS
LIN {X 745.516, Y -389.585, Z 86.15, A 0, B 90, C -0, E1 0, E2 0, E3 0, E4 0} C_DIS
LIN {X 744.216, Y -389.985, Z 86.15, A 0, B 90, C -0, E1 0, E2 0, E3 0, E4 0} C_DIS
LIN {X 737.346, Y -390.588, Z 86.15, A 0, B 90, C -0, E1 0, E2 0, E3 0, E4 0} C_DIS
LIN {X 736.138, Y -391.126, Z 86.15, A 0, B 90, C -0, E1 0, E2 0, E3 0, E4 0} C_DIS
LIN {X 736.134, Y -392.471, Z 86.15, A 0, B 90, C -0, E1 0, E2 0, E3 0, E4 0} C_DIS
LIN {X 737.614, Y -399.206, Z 86.15, A 0, B 90, C -0, E1 0, E2 0, E3 0, E4 0} C_DIS
LIN {X 737.515, Y -400.558, Z 86.15, A 0, B 90, C -0, E1 0, E2 0, E3 0, E4 0} C_DIS
LIN {X 736.59, Y -401.555, Z 86.15, A 0, B 90, C -0, E1 0, E2 0, E3 0, E4 0} C_DIS
LIN {X 730.942, Y -405.512, Z 86.15, A 0, B 90, C -0, E1 0, E2 0, E3 0, E4 0} C_DIS
LIN {X 730.165, Y -406.582, Z 86.15, A 0, B 90, C -0, E1 0, E2 0, E3 0, E4 0} C_DIS
LIN {X 730.834, Y -407.749, Z 86.15, A 0, B 90, C -0, E1 0, E2 0, E3 0, E4 0} C_DIS
LIN {X 735.483, Y -412.842, Z 86.15, A 0, B 90, C -0, E1 0, E2 0, E3 0, E4 0} C_DIS
LIN {X 736.074, Y -414.062, Z 86.15, A 0, B 90, C -0, E1 0, E2 0, E3 0, E4 0} C_DIS
LIN {X 735.771, Y -415.387, Z 86.15, A 0, B 90, C -0, E1 0, E2 0, E3 0, E4 0} C_DIS
LIN {X 732.858, Y -421.638, Z 86.15, A 0, B 90, C -0, E1 0, E2 0, E3 0, E4 0} C_DIS
LIN {X 732.72, Y -422.953, Z 86.15, A 0, B 90, C -0, E1 0, E2 0, E3 0, E4 0} C_DIS
LIN {X 733.883, Y -423.63, Z 86.15, A 0, B 90, C -0, E1 0, E2 0, E3 0, E4 0} C_DIS
LIN {X 740.456, Y -425.716, Z 86.15, A 0, B 90, C -0, E1 0, E2 0, E3 0, E4 0} C_DIS
LIN {X 741.577, Y -426.477, Z 86.15, A 0, B 90, C -0, E1 0, E2 0, E3 0, E4 0} C_DIS
LIN {X 741.977, Y -427.777, Z 86.15, A 0, B 90, C -0, E1 0, E2 0, E3 0, E4 0} C_DIS
LIN {X 742.58, Y -434.646, Z 86.15, A 0, B 90, C -0, E1 0, E2 0, E3 0, E4 0} C_DIS
LIN {X 743.119, Y -435.854, Z 86.15, A 0, B 90, C -0, E1 0, E2 0, E3 0, E4 0} C_DIS
LIN {X 744.464, Y -435.859, Z 86.15, A 0, B 90, C -0, E1 0, E2 0, E3 0, E4 0} C_DIS
LIN {X 751.199, Y -434.378, Z 86.15, A 0, B 90, C -0, E1 0, E2 0, E3 0, E4 0} C_DIS
LIN {X 752.551, Y -434.477, Z 86.15, A 0, B 90, C -0, E1 0, E2 0, E3 0, E4 0} C_DIS
LIN {X 753.547, Y -435.402, Z 86.15, A 0, B 90, C -0, E1 0, E2 0, E3 0, E4 0} C_DIS
LIN {X 757.504, Y -441.05, Z 86.15, A 0, B 90, C -0, E1 0, E2 0, E3 0, E4 0} C_DIS
LIN {X 758.574, Y -441.827, Z 86.15, A 0, B 90, C -0, E1 0, E2 0, E3 0, E4 0} C_DIS
LIN {X 759.741, Y -441.159, Z 86.15, A 0, B 90, C -0, E1 0, E2 0, E3 0, E4 0} C_DIS
LIN {X 764.834, Y -436.509, Z 86.15, A 0, B 90, C -0, E1 0, E2 0, E3 0, E4 0} C_DIS
LIN {X 766.054, Y -435.919, Z 86.15, A 0, B 90, C -0, E1 0, E2 0, E3 0, E4 0} C_DIS
LIN {X 767.38, Y -436.222, Z 86.15, A 0, B 90, C -0, E1 0, E2 0, E3 0, E4 0} C_DIS
LIN {X 773.631, Y -439.135, Z 86.15, A 0, B 90, C -0, E1 0, E2 0, E3 0, E4 0} C_DIS
LIN {X 774.946, Y -439.272, Z 86.15, A 0, B 90, C -0, E1 0, E2 0, E3 0, E4 0} C_DIS
LIN {X 775.622, Y -438.11, Z 86.15, A 0, B 90, C -0, E1 0, E2 0, E3 0, E4 0} C_DIS
LIN {X 777.708, Y -431.537, Z 86.15, A 0, B 90, C -0, E1 0, E2 0, E3 0, E4 0} C_DIS
LIN {X 778.469, Y -430.415, Z 86.15, A 0, B 90, C -0, E1 0, E2 0, E3 0, E4 0} C_DIS
LIN {X 779.769, Y -430.015, Z 86.15, A 0, B 90, C -0, E1 0, E2 0, E3 0, E4 0} C_DIS
LIN {X 786.639, Y -429.412, Z 86.15, A 0, B 90, C -0, E1 0, E2 0, E3 0, E4 0} C_DIS
LIN {X 787.847, Y -428.874, Z 86.15, A 0, B 90, C -0, E1 0, E2 0, E3 0, E4 0} C_DIS
LIN {X 787.851, Y -427.529, Z 86.15, A 0, B 90, C -0, E1 0, E2 0, E3 0, E4 0} C_DIS
LIN {X 786.371, Y -420.794, Z 86.15, A 0, B 90, C -0, E1 0, E2 0, E3 0, E4 0} C_DIS
LIN {X 786.469, Y -419.442, Z 86.15, A 0, B 90, C -0, E1 0, E2 0, E3 0, E4 0} C_DIS
LIN {X 787.395, Y -418.445, Z 86.15, A 0, B 90, C -0, E1 0, E2 0, E3 0, E4 0} C_DIS
LIN {X 793.043, Y -414.488, Z 86.15, A 0, B 90, C -0, E1 0, E2 0, E3 0, E4 0} C_DIS
LIN {X 793.82, Y -413.418, Z 86.15, A 0, B 90, C -0, E1 0, E2 0, E3 0, E4 0} C_DIS
LIN {X 793.151, Y -412.251, Z 86.15, A 0, B 90, C -0, E1 0, E2 0, E3 0, E4 0} C_DIS
LIN {X 788.502, Y -407.158, Z 86.15, A 0, B 90, C -0, E1 0, E2 0, E3 0, E4 0} C_DIS
LIN {X 787.911, Y -405.938, Z 86.15, A 0, B 90, C -0, E1 0, E2 0, E3 0, E4 0} C_DIS
LIN {X 788.214, Y -404.613, Z 86.15, A 0, B 90, C -0, E1 0, E2 0, E3 0, E4 0} C_DIS
LIN {X 791.127, Y -398.362, Z 86.15, A 0, B 90, C -0, E1 0, E2 0, E3 0, E4 0} C_DIS
LIN {X 791.265, Y -397.047, Z 86.15, A 0, B 90, C -0, E1 0, E2 0, E3 0, E4 0} C_DIS
LIN {X 790.102, Y -396.37, Z 86.15, A 0, B 90, C -0, E1 0, E2 0, E3 0, E4 0} C_DIS
LIN {X 783.529, Y -394.284, Z 86.15, A 0, B 90, C -0, E1 0, E2 0, E3 0, E4 0} C_DIS
LIN {X 782.408, Y -393.523, Z 86.15, A 0, B 90, C -0, E1 0, E2 0, E3 0, E4 0} C_DIS
LIN {X 782.008, Y -392.223, Z 86.15, A 0, B 90, C -0, E1 0, E2 0, E3 0, E4 0} C_DIS
LIN {X 781.405, Y -385.354, Z 86.15, A 0, B 90, C -0, E1 0, E2 0, E3 0, E4 0} C_DIS
LIN {X 780.866, Y -384.146, Z 86.15, A 0, B 90, C -0, E1 0, E2 0, E3 0, E4 0} C_DIS
LIN {X 779.521, Y -384.141, Z 86.15, A 0, B 90, C -0, E1 0, E2 0, E3 0, E4 0} C_DIS
LIN {X 774.133, Y -385.326, Z 86.15, A 0, B 90, C -0, E1 0, E2 0, E3 0, E4 0} C_DIS
LIN {X 772.517, Y -385.666, Z 86.8, A 0, B 90, C -0, E1 0, E2 0, E3 0, E4 0} C_DIS
LIN {X 771.172, Y -385.579, Z 86.8, A 0, B 90, C -0, E1 0, E2 0, E3 0, E4 0} C_DIS
LIN {X 770.173, Y -384.667, Z 86.8, A 0, B 90, C -0, E1 0, E2 0, E3 0, E4 0} C_DIS
LIN {X 766.19, Y -379.085, Z 86.8, A 0, B 90, C -0, E1 0, E2 0, E3 0, E4 0} C_DIS
LIN {X 765.12, Y -378.322, Z 86.8, A 0, B 90, C -0, E1 0, E2 0, E3 0, E4 0} C_DIS
LIN {X 763.965, Y -378.996, Z 86.8, A 0, B 90, C -0, E1 0, E2 0, E3 0, E4 0} C_DIS
LIN {X 758.94, Y -383.663, Z 86.8, A 0, B 90, C -0, E1 0, E2 0, E3 0, E4 0} C_DIS
LIN {X 757.732, Y -384.261, Z 86.8, A 0, B 90, C -0, E1 0, E2 0, E3 0, E4 0} C_DIS
LIN {X 756.411, Y -383.971, Z 86.8, A 0, B 90, C -0, E1 0, E2 0, E3 0, E4 0} C_DIS
LIN {X 750.17, Y -381.128, Z 86.8, A 0, B 90, C -0, E1 0, E2 0, E3 0, E4 0} C_DIS
LIN {X 748.861, Y -381.002, Z 86.8, A 0, B 90, C -0, E1 0, E2 0, E3 0, E4 0} C_DIS
LIN {X 748.198, Y -382.164, Z 86.8, A 0, B 90, C -0, E1 0, E2 0, E3 0, E4 0} C_DIS
LIN {X 746.181, Y -388.718, Z 86.8, A 0, B 90, C -0, E1 0, E2 0, E3 0, E4 0} C_DIS
LIN {X 745.433, Y -389.84, Z 86.8, A 0, B 90, C -0, E1 0, E2 0, E3 0, E4 0} C_DIS
LIN {X 744.144, Y -390.249, Z 86.8, A 0, B 90, C -0, E1 0, E2 0, E3 0, E4 0} C_DIS
LIN {X 737.318, Y -390.907, Z 86.8, A 0, B 90, C -0, E1 0, E2 0, E3 0, E4 0} C_DIS
LIN {X 736.122, Y -391.453, Z 86.8, A 0, B 90, C -0, E1 0, E2 0, E3 0, E4 0} C_DIS
LIN {X 736.128, Y -392.79, Z 86.8, A 0, B 90, C -0, E1 0, E2 0, E3 0, E4 0} C_DIS
LIN {X 737.658, Y -399.475, Z 86.8, A 0, B 90, C -0, E1 0, E2 0, E3 0, E4 0} C_DIS
LIN {X 737.572, Y -400.82, Z 86.8, A 0, B 90, C -0, E1 0, E2 0, E3 0, E4 0} C_DIS
LIN {X 736.66, Y -401.819, Z 86.8, A 0, B 90, C -0, E1 0, E2 0, E3 0, E4 0} C_DIS
LIN {X 731.077, Y -405.802, Z 86.8, A 0, B 90, C -0, E1 0, E2 0, E3 0, E4 0} C_DIS
LIN {X 730.314, Y -406.873, Z 86.8, A 0, B 90, C -0, E1 0, E2 0, E3 0, E4 0} C_DIS
LIN {X 730.989, Y -408.028, Z 86.8, A 0, B 90, C -0, E1 0, E2 0, E3 0, E4 0} C_DIS
LIN {X 735.656, Y -413.052, Z 86.8, A 0, B 90, C -0, E1 0, E2 0, E3 0, E4 0} C_DIS
LIN {X 736.253, Y -414.26, Z 86.8, A 0, B 90, C -0, E1 0, E2 0, E3 0, E4 0} C_DIS
LIN {X 735.963, Y -415.581, Z 86.8, A 0, B 90, C -0, E1 0, E2 0, E3 0, E4 0} C_DIS
LIN {X 733.12, Y -421.822, Z 86.8, A 0, B 90, C -0, E1 0, E2 0, E3 0, E4 0} C_DIS
LIN {X 732.995, Y -423.131, Z 86.8, A 0, B 90, C -0, E1 0, E2 0, E3 0, E4 0} C_DIS
LIN {X 734.156, Y -423.794, Z 86.8, A 0, B 90, C -0, E1 0, E2 0, E3 0, E4 0} C_DIS
LIN {X 740.711, Y -425.812, Z 86.8, A 0, B 90, C -0, E1 0, E2 0, E3 0, E4 0} C_DIS
LIN {X 741.832, Y -426.559, Z 86.8, A 0, B 90, C -0, E1 0, E2 0, E3 0, E4 0} C_DIS
LIN {X 742.241, Y -427.848, Z 86.8, A 0, B 90, C -0, E1 0, E2 0, E3 0, E4 0} C_DIS
LIN {X 742.9, Y -434.674, Z 86.8, A 0, B 90, C -0, E1 0, E2 0, E3 0, E4 0} C_DIS
LIN {X 743.445, Y -435.871, Z 86.8, A 0, B 90, C -0, E1 0, E2 0, E3 0, E4 0} C_DIS
LIN {X 744.783, Y -435.864, Z 86.8, A 0, B 90, C -0, E1 0, E2 0, E3 0, E4 0} C_DIS
LIN {X 751.468, Y -434.334, Z 86.8, A 0, B 90, C -0, E1 0, E2 0, E3 0, E4 0} C_DIS
LIN {X 752.813, Y -434.421, Z 86.8, A 0, B 90, C -0, E1 0, E2 0, E3 0, E4 0} C_DIS
LIN {X 753.812, Y -435.333, Z 86.8, A 0, B 90, C -0, E1 0, E2 0, E3 0, E4 0} C_DIS
LIN {X 757.795, Y -440.915, Z 86.8, A 0, B 90, C -0, E1 0, E2 0, E3 0, E4 0} C_DIS
LIN {X 758.865, Y -441.678, Z 86.8, A 0, B 90, C -0, E1 0, E2 0, E3 0, E4 0} C_DIS
LIN {X 760.02, Y -441.004, Z 86.8, A 0, B 90, C -0, E1 0, E2 0, E3 0, E4 0} C_DIS
LIN {X 765.045, Y -436.337, Z 86.8, A 0, B 90, C -0, E1 0, E2 0, E3 0, E4 0} C_DIS
LIN {X 766.253, Y -435.739, Z 86.8, A 0, B 90, C -0, E1 0, E2 0, E3 0, E4 0} C_DIS
LIN {X 767.574, Y -436.029, Z 86.8, A 0, B 90, C -0, E1 0, E2 0, E3 0, E4 0} C_DIS
LIN {X 773.815, Y -438.872, Z 86.8, A 0, B 90, C -0, E1 0, E2 0, E3 0, E4 0} C_DIS
LIN {X 775.124, Y -438.998, Z 86.8, A 0, B 90, C -0, E1 0, E2 0, E3 0, E4 0} C_DIS
LIN {X 775.786, Y -437.836, Z 86.8, A 0, B 90, C -0, E1 0, E2 0, E3 0, E4 0} C_DIS
LIN {X 777.804, Y -431.282, Z 86.8, A 0, B 90, C -0, E1 0, E2 0, E3 0, E4 0} C_DIS
LIN {X 778.552, Y -430.16, Z 86.8, A 0, B 90, C -0, E1 0, E2 0, E3 0, E4 0} C_DIS
LIN {X 779.841, Y -429.751, Z 86.8, A 0, B 90, C -0, E1 0, E2 0, E3 0, E4 0} C_DIS
LIN {X 786.667, Y -429.093, Z 86.8, A 0, B 90, C -0, E1 0, E2 0, E3 0, E4 0} C_DIS
LIN {X 787.863, Y -428.547, Z 86.8, A 0, B 90, C -0, E1 0, E2 0, E3 0, E4 0} C_DIS
LIN {X 787.857, Y -427.21, Z 86.8, A 0, B 90, C -0, E1 0, E2 0, E3 0, E4 0} C_DIS
LIN {X 786.327, Y -420.525, Z 86.8, A 0, B 90, C -0, E1 0, E2 0, E3 0, E4 0} C_DIS
LIN {X 786.413, Y -419.18, Z 86.8, A 0, B 90, C -0, E1 0, E2 0, E3 0, E4 0} C_DIS
LIN {X 787.325, Y -418.181, Z 86.8, A 0, B 90, C -0, E1 0, E2 0, E3 0, E4 0} C_DIS
LIN {X 792.908, Y -414.198, Z 86.8, A 0, B 90, C -0, E1 0, E2 0, E3 0, E4 0} C_DIS
LIN {X 793.671, Y -413.127, Z 86.8, A 0, B 90, C -0, E1 0, E2 0, E3 0, E4 0} C_DIS
LIN {X 792.996, Y -411.972, Z 86.8, A 0, B 90, C -0, E1 0, E2 0, E3 0, E4 0} C_DIS
LIN {X 788.329, Y -406.948, Z 86.8, A 0, B 90, C -0, E1 0, E2 0, E3 0, E4 0} C_DIS
LIN {X 787.732, Y -405.74, Z 86.8, A 0, B 90, C -0, E1 0, E2 0, E3 0, E4 0} C_DIS
LIN {X 788.022, Y -404.419, Z 86.8, A 0, B 90, C -0, E1 0, E2 0, E3 0, E4 0} C_DIS
LIN {X 790.865, Y -398.178, Z 86.8, A 0, B 90, C -0, E1 0, E2 0, E3 0, E4 0} C_DIS
LIN {X 790.99, Y -396.869, Z 86.8, A 0, B 90, C -0, E1 0, E2 0, E3 0, E4 0} C_DIS
LIN {X 789.829, Y -396.206, Z 86.8, A 0, B 90, C -0, E1 0, E2 0, E3 0, E4 0} C_DIS
LIN {X 783.274, Y -394.188, Z 86.8, A 0, B 90, C -0, E1 0, E2 0, E3 0, E4 0} C_DIS
LIN {X 782.153, Y -393.441, Z 86.8, A 0, B 90, C -0, E1 0, E2 0, E3 0, E4 0} C_DIS
LIN {X 781.744, Y -392.152, Z 86.8, A 0, B 90, C -0, E1 0, E2 0, E3 0, E4 0} C_DIS
LIN {X 781.085, Y -385.326, Z 86.8, A 0, B 90, C -0, E1 0, E2 0, E3 0, E4 0} C_DIS
LIN {X 780.54, Y -384.129, Z 86.8, A 0, B 90, C -0, E1 0, E2 0, E3 0, E4 0} C_DIS
LIN {X 779.202, Y -384.136, Z 86.8, A 0, B 90, C -0, E1 0, E2 0, E3 0, E4 0} C_DIS
LIN {X 773.854, Y -385.36, Z 86.8, A 0, B 90, C -0, E1 0, E2 0, E3 0, E4 0} C_DIS
LIN {X 772.251, Y -385.711, Z 87.45, A 0, B 90, C -0, E1 0, E2 0, E3 0, E4 0} C_DIS
LIN {X 770.913, Y -385.636, Z 87.45, A 0, B 90, C -0, E1 0, E2 0, E3 0, E4 0} C_DIS
LIN {X 769.912, Y -384.738, Z 87.45, A 0, B 90, C -0, E1 0, E2 0, E3 0, E4 0} C_DIS
LIN {X 765.903, Y -379.221, Z 87.45, A 0, B 90, C -0, E1 0, E2 0, E3 0, E4 0} C_DIS
LIN {X 764.832, Y -378.471, Z 87.45, A 0, B 90, C -0, E1 0, E2 0, E3 0, E4 0} C_DIS
LIN {X 763.689, Y -379.151, Z 87.45, A 0, B 90, C -0, E1 0, E2 0, E3 0, E4 0} C_DIS
LIN {X 758.732, Y -383.836, Z 87.45, A 0, B 90, C -0, E1 0, E2 0, E3 0, E4 0} C_DIS
LIN {X 757.536, Y -384.44, Z 87.45, A 0, B 90, C -0, E1 0, E2 0, E3 0, E4 0} C_DIS
LIN {X 756.22, Y -384.163, Z 87.45, A 0, B 90, C -0, E1 0, E2 0, E3 0, E4 0} C_DIS
LIN {X 749.99, Y -381.389, Z 87.45, A 0, B 90, C -0, E1 0, E2 0, E3 0, E4 0} C_DIS
LIN {X 748.687, Y -381.275, Z 87.45, A 0, B 90, C -0, E1 0, E2 0, E3 0, E4 0} C_DIS
LIN {X 748.038, Y -382.436, Z 87.45, A 0, B 90, C -0, E1 0, E2 0, E3 0, E4 0} C_DIS
LIN {X 746.087, Y -388.971, Z 87.45, A 0, B 90, C -0, E1 0, E2 0, E3 0, E4 0} C_DIS
LIN {X 745.353, Y -390.093, Z 87.45, A 0, B 90, C -0, E1 0, E2 0, E3 0, E4 0} C_DIS
LIN {X 744.075, Y -390.511, Z 87.45, A 0, B 90, C -0, E1 0, E2 0, E3 0, E4 0} C_DIS
LIN {X 737.292, Y -391.224, Z 87.45, A 0, B 90, C -0, E1 0, E2 0, E3 0, E4 0} C_DIS
LIN {X 736.107, Y -391.776, Z 87.45, A 0, B 90, C -0, E1 0, E2 0, E3 0, E4 0} C_DIS
LIN {X 736.125, Y -393.106, Z 87.45, A 0, B 90, C -0, E1 0, E2 0, E3 0, E4 0} C_DIS
LIN {X 737.703, Y -399.741, Z 87.45, A 0, B 90, C -0, E1 0, E2 0, E3 0, E4 0} C_DIS
LIN {X 737.629, Y -401.079, Z 87.45, A 0, B 90, C -0, E1 0, E2 0, E3 0, E4 0} C_DIS
LIN {X 736.731, Y -402.081, Z 87.45, A 0, B 90, C -0, E1 0, E2 0, E3 0, E4 0} C_DIS
LIN {X 731.213, Y -406.089, Z 87.45, A 0, B 90, C -0, E1 0, E2 0, E3 0, E4 0} C_DIS
LIN {X 730.463, Y -407.161, Z 87.45, A 0, B 90, C -0, E1 0, E2 0, E3 0, E4 0} C_DIS
LIN {X 731.144, Y -408.303, Z 87.45, A 0, B 90, C -0, E1 0, E2 0, E3 0, E4 0} C_DIS
LIN {X 735.828, Y -413.26, Z 87.45, A 0, B 90, C -0, E1 0, E2 0, E3 0, E4 0} C_DIS
LIN {X 736.433, Y -414.456, Z 87.45, A 0, B 90, C -0, E1 0, E2 0, E3 0, E4 0} C_DIS
LIN {X 736.155, Y -415.772, Z 87.45, A 0, B 90, C -0, E1 0, E2 0, E3 0, E4 0} C_DIS
LIN {X 733.381, Y -422.003, Z 87.45, A 0, B 90, C -0, E1 0, E2 0, E3 0, E4 0} C_DIS
LIN {X 733.268, Y -423.306, Z 87.45, A 0, B 90, C -0, E1 0, E2 0, E3 0, E4 0} C_DIS
LIN {X 734.428, Y -423.955, Z 87.45, A 0, B 90, C -0, E1 0, E2 0, E3 0, E4 0} C_DIS
LIN {X 740.964, Y -425.906, Z 87.45, A 0, B 90, C -0, E1 0, E2 0, E3 0, E4 0} C_DIS
LIN {X 742.085, Y -426.639, Z 87.45, A 0, B 90, C -0, E1 0, E2 0, E3 0, E4 0} C_DIS
LIN {X 742.503, Y -427.918, Z 87.45, A 0, B 90, C -0, E1 0, E2 0, E3 0, E4 0} C_DIS
LIN {X 743.216, Y -434.7, Z 87.45, A 0, B 90, C -0, E1 0, E2 0, E3 0, E4 0} C_DIS
LIN {X 743.769, Y -435.885, Z 87.45, A 0, B 90, C -0, E1 0, E2 0, E3 0, E4 0} C_DIS
LIN {X 745.099, Y -435.867, Z 87.45, A 0, B 90, C -0, E1 0, E2 0, E3 0, E4 0} C_DIS
LIN {X 751.734, Y -434.289, Z 87.45, A 0, B 90, C -0, E1 0, E2 0, E3 0, E4 0} C_DIS
LIN {X 753.072, Y -434.364, Z 87.45, A 0, B 90, C -0, E1 0, E2 0, E3 0, E4 0} C_DIS
LIN {X 754.073, Y -435.262, Z 87.45, A 0, B 90, C -0, E1 0, E2 0, E3 0, E4 0} C_DIS
LIN {X 758.082, Y -440.779, Z 87.45, A 0, B 90, C -0, E1 0, E2 0, E3 0, E4 0} C_DIS
LIN {X 759.153, Y -441.529, Z 87.45, A 0, B 90, C -0, E1 0, E2 0, E3 0, E4 0} C_DIS
LIN {X 760.296, Y -440.849, Z 87.45, A 0, B 90, C -0, E1 0, E2 0, E3 0, E4 0} C_DIS
LIN {X 765.253, Y -436.164, Z 87.45, A 0, B 90, C -0, E1 0, E2 0, E3 0, E4 0} C_DIS
LIN {X 766.449, Y -435.56, Z 87.45, A 0, B 90, C -0, E1 0, E2 0, E3 0, E4 0} C_DIS
LIN {X 767.765, Y -435.837, Z 87.45, A 0, B 90, C -0, E1 0, E2 0, E3 0, E4 0} C_DIS
LIN {X 773.995, Y -438.611, Z 87.45, A 0, B 90, C -0, E1 0, E2 0, E3 0, E4 0} C_DIS
LIN {X 775.298, Y -438.725, Z 87.45, A 0, B 90, C -0, E1 0, E2 0, E3 0, E4 0} C_DIS
LIN {X 775.947, Y -437.564, Z 87.45, A 0, B 90, C -0, E1 0, E2 0, E3 0, E4 0} C_DIS
LIN {X 777.898, Y -431.029, Z 87.45, A 0, B 90, C -0, E1 0, E2 0, E3 0, E4 0} C_DIS
LIN {X 778.632, Y -429.907, Z 87.45, A 0, B 90, C -0, E1 0, E2 0, E3 0, E4 0} C_DIS
LIN {X 779.91, Y -429.489, Z 87.45, A 0, B 90, C -0, E1 0, E2 0, E3 0, E4 0} C_DIS
LIN {X 786.693, Y -428.776, Z 87.45, A 0, B 90, C -0, E1 0, E2 0, E3 0, E4 0} C_DIS
LIN {X 787.878, Y -428.224, Z 87.45, A 0, B 90, C -0, E1 0, E2 0, E3 0, E4 0} C_DIS
LIN {X 787.86, Y -426.894, Z 87.45, A 0, B 90, C -0, E1 0, E2 0, E3 0, E4 0} C_DIS
LIN {X 786.282, Y -420.259, Z 87.45, A 0, B 90, C -0, E1 0, E2 0, E3 0, E4 0} C_DIS
LIN {X 786.356, Y -418.921, Z 87.45, A 0, B 90, C -0, E1 0, E2 0, E3 0, E4 0} C_DIS
LIN {X 787.254, Y -417.919, Z 87.45, A 0, B 90, C -0, E1 0, E2 0, E3 0, E4 0} C_DIS
LIN {X 792.772, Y -413.911, Z 87.45, A 0, B 90, C -0, E1 0, E2 0, E3 0, E4 0} C_DIS
LIN {X 793.522, Y -412.839, Z 87.45, A 0, B 90, C -0, E1 0, E2 0, E3 0, E4 0} C_DIS
LIN {X 792.841, Y -411.697, Z 87.45, A 0, B 90, C -0, E1 0, E2 0, E3 0, E4 0} C_DIS
LIN {X 788.157, Y -406.74, Z 87.45, A 0, B 90, C -0, E1 0, E2 0, E3 0, E4 0} C_DIS
LIN {X 787.552, Y -405.544, Z 87.45, A 0, B 90, C -0, E1 0, E2 0, E3 0, E4 0} C_DIS
LIN {X 787.83, Y -404.228, Z 87.45, A 0, B 90, C -0, E1 0, E2 0, E3 0, E4 0} C_DIS
LIN {X 790.604, Y -397.997, Z 87.45, A 0, B 90, C -0, E1 0, E2 0, E3 0, E4 0} C_DIS
LIN {X 790.717, Y -396.694, Z 87.45, A 0, B 90, C -0, E1 0, E2 0, E3 0, E4 0} C_DIS
LIN {X 789.557, Y -396.045, Z 87.45, A 0, B 90, C -0, E1 0, E2 0, E3 0, E4 0} C_DIS
LIN {X 783.021, Y -394.094, Z 87.45, A 0, B 90, C -0, E1 0, E2 0, E3 0, E4 0} C_DIS
LIN {X 781.9, Y -393.361, Z 87.45, A 0, B 90, C -0, E1 0, E2 0, E3 0, E4 0} C_DIS
LIN {X 781.482, Y -392.082, Z 87.45, A 0, B 90, C -0, E1 0, E2 0, E3 0, E4 0} C_DIS
LIN {X 780.769, Y -385.3, Z 87.45, A 0, B 90, C -0, E1 0, E2 0, E3 0, E4 0} C_DIS
LIN {X 780.216, Y -384.115, Z 87.45, A 0, B 90, C -0, E1 0, E2 0, E3 0, E4 0} C_DIS
LIN {X 778.886, Y -384.133, Z 87.45, A 0, B 90, C -0, E1 0, E2 0, E3 0, E4 0} C_DIS
LIN {X 773.578, Y -385.395, Z 87.45, A 0, B 90, C -0, E1 0, E2 0, E3 0, E4 0} C_DIS
LIN {X 771.988, Y -385.757, Z 88.1, A 0, B 90, C -0, E1 0, E2 0, E3 0, E4 0} C_DIS
LIN {X 770.657, Y -385.695, Z 88.1, A 0, B 90, C -0, E1 0, E2 0, E3 0, E4 0} C_DIS
LIN {X 769.653, Y -384.81, Z 88.1, A 0, B 90, C -0, E1 0, E2 0, E3 0, E4 0} C_DIS
LIN {X 765.62, Y -379.357, Z 88.1, A 0, B 90, C -0, E1 0, E2 0, E3 0, E4 0} C_DIS
LIN {X 764.548, Y -378.62, Z 88.1, A 0, B 90, C -0, E1 0, E2 0, E3 0, E4 0} C_DIS
LIN {X 763.417, Y -379.307, Z 88.1, A 0, B 90, C -0, E1 0, E2 0, E3 0, E4 0} C_DIS
LIN {X 758.528, Y -384.007, Z 88.1, A 0, B 90, C -0, E1 0, E2 0, E3 0, E4 0} C_DIS
LIN {X 757.343, Y -384.619, Z 88.1, A 0, B 90, C -0, E1 0, E2 0, E3 0, E4 0} C_DIS
LIN {X 756.032, Y -384.354, Z 88.1, A 0, B 90, C -0, E1 0, E2 0, E3 0, E4 0} C_DIS
LIN {X 749.812, Y -381.649, Z 88.1, A 0, B 90, C -0, E1 0, E2 0, E3 0, E4 0} C_DIS
LIN {X 748.516, Y -381.546, Z 88.1, A 0, B 90, C -0, E1 0, E2 0, E3 0, E4 0} C_DIS
LIN {X 747.88, Y -382.706, Z 88.1, A 0, B 90, C -0, E1 0, E2 0, E3 0, E4 0} C_DIS
LIN {X 745.995, Y -389.222, Z 88.1, A 0, B 90, C -0, E1 0, E2 0, E3 0, E4 0} C_DIS
LIN {X 745.275, Y -390.344, Z 88.1, A 0, B 90, C -0, E1 0, E2 0, E3 0, E4 0} C_DIS
LIN {X 744.008, Y -390.77, Z 88.1, A 0, B 90, C -0, E1 0, E2 0, E3 0, E4 0} C_DIS
LIN {X 737.268, Y -391.537, Z 88.1, A 0, B 90, C -0, E1 0, E2 0, E3 0, E4 0} C_DIS
LIN {X 736.094, Y -392.097, Z 88.1, A 0, B 90, C -0, E1 0, E2 0, E3 0, E4 0} C_DIS
LIN {X 736.124, Y -393.419, Z 88.1, A 0, B 90, C -0, E1 0, E2 0, E3 0, E4 0} C_DIS
LIN {X 737.75, Y -400.004, Z 88.1, A 0, B 90, C -0, E1 0, E2 0, E3 0, E4 0} C_DIS
LIN {X 737.687, Y -401.336, Z 88.1, A 0, B 90, C -0, E1 0, E2 0, E3 0, E4 0} C_DIS
LIN {X 736.802, Y -402.339, Z 88.1, A 0, B 90, C -0, E1 0, E2 0, E3 0, E4 0} C_DIS
LIN {X 731.349, Y -406.373, Z 88.1, A 0, B 90, C -0, E1 0, E2 0, E3 0, E4 0} C_DIS
LIN {X 730.613, Y -407.445, Z 88.1, A 0, B 90, C -0, E1 0, E2 0, E3 0, E4 0} C_DIS
LIN {X 731.299, Y -408.575, Z 88.1, A 0, B 90, C -0, E1 0, E2 0, E3 0, E4 0} C_DIS
LIN {X 736, Y -413.465, Z 88.1, A 0, B 90, C -0, E1 0, E2 0, E3 0, E4 0} C_DIS
LIN {X 736.611, Y -414.649, Z 88.1, A 0, B 90, C -0, E1 0, E2 0, E3 0, E4 0} C_DIS
LIN {X 736.347, Y -415.961, Z 88.1, A 0, B 90, C -0, E1 0, E2 0, E3 0, E4 0} C_DIS
LIN {X 733.641, Y -422.18, Z 88.1, A 0, B 90, C -0, E1 0, E2 0, E3 0, E4 0} C_DIS
LIN {X 733.539, Y -423.477, Z 88.1, A 0, B 90, C -0, E1 0, E2 0, E3 0, E4 0} C_DIS
LIN {X 734.699, Y -424.113, Z 88.1, A 0, B 90, C -0, E1 0, E2 0, E3 0, E4 0} C_DIS
LIN {X 741.215, Y -425.997, Z 88.1, A 0, B 90, C -0, E1 0, E2 0, E3 0, E4 0} C_DIS
LIN {X 742.336, Y -426.717, Z 88.1, A 0, B 90, C -0, E1 0, E2 0, E3 0, E4 0} C_DIS
LIN {X 742.763, Y -427.985, Z 88.1, A 0, B 90, C -0, E1 0, E2 0, E3 0, E4 0} C_DIS
LIN {X 743.53, Y -434.724, Z 88.1, A 0, B 90, C -0, E1 0, E2 0, E3 0, E4 0} C_DIS
LIN {X 744.089, Y -435.898, Z 88.1, A 0, B 90, C -0, E1 0, E2 0, E3 0, E4 0} C_DIS
LIN {X 745.412, Y -435.869, Z 88.1, A 0, B 90, C -0, E1 0, E2 0, E3 0, E4 0} C_DIS
LIN {X 751.997, Y -434.243, Z 88.1, A 0, B 90, C -0, E1 0, E2 0, E3 0, E4 0} C_DIS
LIN {X 753.328, Y -434.305, Z 88.1, A 0, B 90, C -0, E1 0, E2 0, E3 0, E4 0} C_DIS
LIN {X 754.332, Y -435.19, Z 88.1, A 0, B 90, C -0, E1 0, E2 0, E3 0, E4 0} C_DIS
LIN {X 758.365, Y -440.643, Z 88.1, A 0, B 90, C -0, E1 0, E2 0, E3 0, E4 0} C_DIS
LIN {X 759.437, Y -441.38, Z 88.1, A 0, B 90, C -0, E1 0, E2 0, E3 0, E4 0} C_DIS
LIN {X 760.568, Y -440.693, Z 88.1, A 0, B 90, C -0, E1 0, E2 0, E3 0, E4 0} C_DIS
LIN {X 765.457, Y -435.993, Z 88.1, A 0, B 90, C -0, E1 0, E2 0, E3 0, E4 0} C_DIS
LIN {X 766.642, Y -435.381, Z 88.1, A 0, B 90, C -0, E1 0, E2 0, E3 0, E4 0} C_DIS
LIN {X 767.953, Y -435.646, Z 88.1, A 0, B 90, C -0, E1 0, E2 0, E3 0, E4 0} C_DIS
LIN {X 774.173, Y -438.351, Z 88.1, A 0, B 90, C -0, E1 0, E2 0, E3 0, E4 0} C_DIS
LIN {X 775.469, Y -438.454, Z 88.1, A 0, B 90, C -0, E1 0, E2 0, E3 0, E4 0} C_DIS
LIN {X 776.105, Y -437.294, Z 88.1, A 0, B 90, C -0, E1 0, E2 0, E3 0, E4 0} C_DIS
LIN {X 777.99, Y -430.778, Z 88.1, A 0, B 90, C -0, E1 0, E2 0, E3 0, E4 0} C_DIS
LIN {X 778.71, Y -429.656, Z 88.1, A 0, B 90, C -0, E1 0, E2 0, E3 0, E4 0} C_DIS
LIN {X 779.977, Y -429.23, Z 88.1, A 0, B 90, C -0, E1 0, E2 0, E3 0, E4 0} C_DIS
LIN {X 786.717, Y -428.463, Z 88.1, A 0, B 90, C -0, E1 0, E2 0, E3 0, E4 0} C_DIS
LIN {X 787.891, Y -427.903, Z 88.1, A 0, B 90, C -0, E1 0, E2 0, E3 0, E4 0} C_DIS
LIN {X 787.861, Y -426.581, Z 88.1, A 0, B 90, C -0, E1 0, E2 0, E3 0, E4 0} C_DIS
LIN {X 786.235, Y -419.996, Z 88.1, A 0, B 90, C -0, E1 0, E2 0, E3 0, E4 0} C_DIS
LIN {X 786.298, Y -418.664, Z 88.1, A 0, B 90, C -0, E1 0, E2 0, E3 0, E4 0} C_DIS
LIN {X 787.183, Y -417.661, Z 88.1, A 0, B 90, C -0, E1 0, E2 0, E3 0, E4 0} C_DIS
LIN {X 792.636, Y -413.627, Z 88.1, A 0, B 90, C -0, E1 0, E2 0, E3 0, E4 0} C_DIS
LIN {X 793.372, Y -412.555, Z 88.1, A 0, B 90, C -0, E1 0, E2 0, E3 0, E4 0} C_DIS
LIN {X 792.686, Y -411.425, Z 88.1, A 0, B 90, C -0, E1 0, E2 0, E3 0, E4 0} C_DIS
LIN {X 787.985, Y -406.535, Z 88.1, A 0, B 90, C -0, E1 0, E2 0, E3 0, E4 0} C_DIS
LIN {X 787.374, Y -405.351, Z 88.1, A 0, B 90, C -0, E1 0, E2 0, E3 0, E4 0} C_DIS
LIN {X 787.638, Y -404.039, Z 88.1, A 0, B 90, C -0, E1 0, E2 0, E3 0, E4 0} C_DIS
LIN {X 790.344, Y -397.82, Z 88.1, A 0, B 90, C -0, E1 0, E2 0, E3 0, E4 0} C_DIS
LIN {X 790.446, Y -396.523, Z 88.1, A 0, B 90, C -0, E1 0, E2 0, E3 0, E4 0} C_DIS
LIN {X 789.286, Y -395.887, Z 88.1, A 0, B 90, C -0, E1 0, E2 0, E3 0, E4 0} C_DIS
LIN {X 782.77, Y -394.003, Z 88.1, A 0, B 90, C -0, E1 0, E2 0, E3 0, E4 0} C_DIS
LIN {X 781.648, Y -393.283, Z 88.1, A 0, B 90, C -0, E1 0, E2 0, E3 0, E4 0} C_DIS
LIN {X 781.222, Y -392.015, Z 88.1, A 0, B 90, C -0, E1 0, E2 0, E3 0, E4 0} C_DIS
LIN {X 780.455, Y -385.276, Z 88.1, A 0, B 90, C -0, E1 0, E2 0, E3 0, E4 0} C_DIS
LIN {X 779.896, Y -384.102, Z 88.1, A 0, B 90, C -0, E1 0, E2 0, E3 0, E4 0} C_DIS
LIN {X 778.573, Y -384.131, Z 88.1, A 0, B 90, C -0, E1 0, E2 0, E3 0, E4 0} C_DIS
LIN {X 773.305, Y -385.432, Z 88.1, A 0, B 90, C -0, E1 0, E2 0, E3 0, E4 0} C_DIS
LIN {X 771.728, Y -385.805, Z 88.75, A 0, B 90, C -0, E1 0, E2 0, E3 0, E4 0} C_DIS
LIN {X 770.403, Y -385.754, Z 88.75, A 0, B 90, C -0, E1 0, E2 0, E3 0, E4 0} C_DIS
LIN {X 769.398, Y -384.882, Z 88.75, A 0, B 90, C -0, E1 0, E2 0, E3 0, E4 0} C_DIS
LIN {X 765.34, Y -379.493, Z 88.75, A 0, B 90, C -0, E1 0, E2 0, E3 0, E4 0} C_DIS
LIN {X 764.268, Y -378.77, Z 88.75, A 0, B 90, C -0, E1 0, E2 0, E3 0, E4 0} C_DIS
LIN {X 763.149, Y -379.462, Z 88.75, A 0, B 90, C -0, E1 0, E2 0, E3 0, E4 0} C_DIS
LIN {X 758.326, Y -384.179, Z 88.75, A 0, B 90, C -0, E1 0, E2 0, E3 0, E4 0} C_DIS
LIN {X 757.153, Y -384.797, Z 88.75, A 0, B 90, C -0, E1 0, E2 0, E3 0, E4 0} C_DIS
LIN {X 755.847, Y -384.545, Z 88.75, A 0, B 90, C -0, E1 0, E2 0, E3 0, E4 0} C_DIS
LIN {X 749.638, Y -381.907, Z 88.75, A 0, B 90, C -0, E1 0, E2 0, E3 0, E4 0} C_DIS
LIN {X 748.348, Y -381.816, Z 88.75, A 0, B 90, C -0, E1 0, E2 0, E3 0, E4 0} C_DIS
LIN {X 747.725, Y -382.975, Z 88.75, A 0, B 90, C -0, E1 0, E2 0, E3 0, E4 0} C_DIS
LIN {X 745.906, Y -389.471, Z 88.75, A 0, B 90, C -0, E1 0, E2 0, E3 0, E4 0} C_DIS
LIN {X 745.2, Y -390.593, Z 88.75, A 0, B 90, C -0, E1 0, E2 0, E3 0, E4 0} C_DIS
LIN {X 743.942, Y -391.028, Z 88.75, A 0, B 90, C -0, E1 0, E2 0, E3 0, E4 0} C_DIS
LIN {X 737.246, Y -391.848, Z 88.75, A 0, B 90, C -0, E1 0, E2 0, E3 0, E4 0} C_DIS
LIN {X 736.084, Y -392.415, Z 88.75, A 0, B 90, C -0, E1 0, E2 0, E3 0, E4 0} C_DIS
LIN {X 736.124, Y -393.73, Z 88.75, A 0, B 90, C -0, E1 0, E2 0, E3 0, E4 0} C_DIS
LIN {X 737.797, Y -400.265, Z 88.75, A 0, B 90, C -0, E1 0, E2 0, E3 0, E4 0} C_DIS
LIN {X 737.746, Y -401.59, Z 88.75, A 0, B 90, C -0, E1 0, E2 0, E3 0, E4 0} C_DIS
LIN {X 736.875, Y -402.595, Z 88.75, A 0, B 90, C -0, E1 0, E2 0, E3 0, E4 0} C_DIS
LIN {X 731.486, Y -406.653, Z 88.75, A 0, B 90, C -0, E1 0, E2 0, E3 0, E4 0} C_DIS
LIN {X 730.762, Y -407.725, Z 88.75, A 0, B 90, C -0, E1 0, E2 0, E3 0, E4 0} C_DIS
LIN {X 731.455, Y -408.844, Z 88.75, A 0, B 90, C -0, E1 0, E2 0, E3 0, E4 0} C_DIS
LIN {X 736.171, Y -413.667, Z 88.75, A 0, B 90, C -0, E1 0, E2 0, E3 0, E4 0} C_DIS
LIN {X 736.789, Y -414.84, Z 88.75, A 0, B 90, C -0, E1 0, E2 0, E3 0, E4 0} C_DIS
LIN {X 736.537, Y -416.146, Z 88.75, A 0, B 90, C -0, E1 0, E2 0, E3 0, E4 0} C_DIS
LIN {X 733.899, Y -422.355, Z 88.75, A 0, B 90, C -0, E1 0, E2 0, E3 0, E4 0} C_DIS
LIN {X 733.809, Y -423.645, Z 88.75, A 0, B 90, C -0, E1 0, E2 0, E3 0, E4 0} C_DIS
LIN {X 734.968, Y -424.268, Z 88.75, A 0, B 90, C -0, E1 0, E2 0, E3 0, E4 0} C_DIS
LIN {X 741.464, Y -426.086, Z 88.75, A 0, B 90, C -0, E1 0, E2 0, E3 0, E4 0} C_DIS
LIN {X 742.586, Y -426.793, Z 88.75, A 0, B 90, C -0, E1 0, E2 0, E3 0, E4 0} C_DIS
LIN {X 743.021, Y -428.05, Z 88.75, A 0, B 90, C -0, E1 0, E2 0, E3 0, E4 0} C_DIS
LIN {X 743.84, Y -434.746, Z 88.75, A 0, B 90, C -0, E1 0, E2 0, E3 0, E4 0} C_DIS
LIN {X 744.407, Y -435.909, Z 88.75, A 0, B 90, C -0, E1 0, E2 0, E3 0, E4 0} C_DIS
LIN {X 745.722, Y -435.868, Z 88.75, A 0, B 90, C -0, E1 0, E2 0, E3 0, E4 0} C_DIS
LIN {X 752.257, Y -434.195, Z 88.75, A 0, B 90, C -0, E1 0, E2 0, E3 0, E4 0} C_DIS
LIN {X 753.582, Y -434.246, Z 88.75, A 0, B 90, C -0, E1 0, E2 0, E3 0, E4 0} C_DIS
LIN {X 754.587, Y -435.118, Z 88.75, A 0, B 90, C -0, E1 0, E2 0, E3 0, E4 0} C_DIS
LIN {X 758.645, Y -440.507, Z 88.75, A 0, B 90, C -0, E1 0, E2 0, E3 0, E4 0} C_DIS
LIN {X 759.717, Y -441.23, Z 88.75, A 0, B 90, C -0, E1 0, E2 0, E3 0, E4 0} C_DIS
LIN {X 760.836, Y -440.538, Z 88.75, A 0, B 90, C -0, E1 0, E2 0, E3 0, E4 0} C_DIS
LIN {X 765.659, Y -435.821, Z 88.75, A 0, B 90, C -0, E1 0, E2 0, E3 0, E4 0} C_DIS
LIN {X 766.832, Y -435.203, Z 88.75, A 0, B 90, C -0, E1 0, E2 0, E3 0, E4 0} C_DIS
LIN {X 768.138, Y -435.455, Z 88.75, A 0, B 90, C -0, E1 0, E2 0, E3 0, E4 0} C_DIS
LIN {X 774.347, Y -438.093, Z 88.75, A 0, B 90, C -0, E1 0, E2 0, E3 0, E4 0} C_DIS
LIN {X 775.637, Y -438.184, Z 88.75, A 0, B 90, C -0, E1 0, E2 0, E3 0, E4 0} C_DIS
LIN {X 776.26, Y -437.025, Z 88.75, A 0, B 90, C -0, E1 0, E2 0, E3 0, E4 0} C_DIS
LIN {X 778.079, Y -430.529, Z 88.75, A 0, B 90, C -0, E1 0, E2 0, E3 0, E4 0} C_DIS
LIN {X 778.785, Y -429.407, Z 88.75, A 0, B 90, C -0, E1 0, E2 0, E3 0, E4 0} C_DIS
LIN {X 780.043, Y -428.972, Z 88.75, A 0, B 90, C -0, E1 0, E2 0, E3 0, E4 0} C_DIS
LIN {X 786.739, Y -428.152, Z 88.75, A 0, B 90, C -0, E1 0, E2 0, E3 0, E4 0} C_DIS
LIN {X 787.901, Y -427.585, Z 88.75, A 0, B 90, C -0, E1 0, E2 0, E3 0, E4 0} C_DIS
LIN {X 787.861, Y -426.27, Z 88.75, A 0, B 90, C -0, E1 0, E2 0, E3 0, E4 0} C_DIS
LIN {X 786.188, Y -419.735, Z 88.75, A 0, B 90, C -0, E1 0, E2 0, E3 0, E4 0} C_DIS
LIN {X 786.239, Y -418.41, Z 88.75, A 0, B 90, C -0, E1 0, E2 0, E3 0, E4 0} C_DIS
LIN {X 787.11, Y -417.405, Z 88.75, A 0, B 90, C -0, E1 0, E2 0, E3 0, E4 0} C_DIS
LIN {X 792.499, Y -413.347, Z 88.75, A 0, B 90, C -0, E1 0, E2 0, E3 0, E4 0} C_DIS
LIN {X 793.223, Y -412.275, Z 88.75, A 0, B 90, C -0, E1 0, E2 0, E3 0, E4 0} C_DIS
LIN {X 792.53, Y -411.156, Z 88.75, A 0, B 90, C -0, E1 0, E2 0, E3 0, E4 0} C_DIS
LIN {X 787.814, Y -406.333, Z 88.75, A 0, B 90, C -0, E1 0, E2 0, E3 0, E4 0} C_DIS
LIN {X 787.196, Y -405.16, Z 88.75, A 0, B 90, C -0, E1 0, E2 0, E3 0, E4 0} C_DIS
LIN {X 787.448, Y -403.854, Z 88.75, A 0, B 90, C -0, E1 0, E2 0, E3 0, E4 0} C_DIS
LIN {X 790.086, Y -397.645, Z 88.75, A 0, B 90, C -0, E1 0, E2 0, E3 0, E4 0} C_DIS
LIN {X 790.176, Y -396.355, Z 88.75, A 0, B 90, C -0, E1 0, E2 0, E3 0, E4 0} C_DIS
LIN {X 789.017, Y -395.732, Z 88.75, A 0, B 90, C -0, E1 0, E2 0, E3 0, E4 0} C_DIS
LIN {X 782.521, Y -393.914, Z 88.75, A 0, B 90, C -0, E1 0, E2 0, E3 0, E4 0} C_DIS
LIN {X 781.399, Y -393.207, Z 88.75, A 0, B 90, C -0, E1 0, E2 0, E3 0, E4 0} C_DIS
LIN {X 780.964, Y -391.95, Z 88.75, A 0, B 90, C -0, E1 0, E2 0, E3 0, E4 0} C_DIS
LIN {X 780.145, Y -385.254, Z 88.75, A 0, B 90, C -0, E1 0, E2 0, E3 0, E4 0} C_DIS
LIN {X 779.578, Y -384.091, Z 88.75, A 0, B 90, C -0, E1 0, E2 0, E3 0, E4 0} C_DIS
LIN {X 778.263, Y -384.132, Z 88.75, A 0, B 90, C -0, E1 0, E2 0, E3 0, E4 0} C_DIS
LIN {X 773.035, Y -385.47, Z 88.75, A 0, B 90, C -0, E1 0, E2 0, E3 0, E4 0} C_DIS
LIN {X 771.47, Y -385.853, Z 89.4, A 0, B 90, C -0, E1 0, E2 0, E3 0, E4 0} C_DIS
LIN {X 770.152, Y -385.814, Z 89.4, A 0, B 90, C -0, E1 0, E2 0, E3 0, E4 0} C_DIS
LIN {X 769.145, Y -384.955, Z 89.4, A 0, B 90, C -0, E1 0, E2 0, E3 0, E4 0} C_DIS
LIN {X 765.063, Y -379.63, Z 89.4, A 0, B 90, C -0, E1 0, E2 0, E3 0, E4 0} C_DIS
LIN {X 763.991, Y -378.919, Z 89.4, A 0, B 90, C -0, E1 0, E2 0, E3 0, E4 0} C_DIS
LIN {X 762.884, Y -379.617, Z 89.4, A 0, B 90, C -0, E1 0, E2 0, E3 0, E4 0} C_DIS
LIN {X 758.127, Y -384.349, Z 89.4, A 0, B 90, C -0, E1 0, E2 0, E3 0, E4 0} C_DIS
LIN {X 756.966, Y -384.974, Z 89.4, A 0, B 90, C -0, E1 0, E2 0, E3 0, E4 0} C_DIS
LIN {X 755.664, Y -384.735, Z 89.4, A 0, B 90, C -0, E1 0, E2 0, E3 0, E4 0} C_DIS
LIN {X 749.467, Y -382.163, Z 89.4, A 0, B 90, C -0, E1 0, E2 0, E3 0, E4 0} C_DIS
LIN {X 748.183, Y -382.084, Z 89.4, A 0, B 90, C -0, E1 0, E2 0, E3 0, E4 0} C_DIS
LIN {X 747.573, Y -383.242, Z 89.4, A 0, B 90, C -0, E1 0, E2 0, E3 0, E4 0} C_DIS
LIN {X 745.819, Y -389.719, Z 89.4, A 0, B 90, C -0, E1 0, E2 0, E3 0, E4 0} C_DIS
LIN {X 745.126, Y -390.84, Z 89.4, A 0, B 90, C -0, E1 0, E2 0, E3 0, E4 0} C_DIS
LIN {X 743.879, Y -391.284, Z 89.4, A 0, B 90, C -0, E1 0, E2 0, E3 0, E4 0} C_DIS
LIN {X 737.226, Y -392.156, Z 89.4, A 0, B 90, C -0, E1 0, E2 0, E3 0, E4 0} C_DIS
LIN {X 736.075, Y -392.729, Z 89.4, A 0, B 90, C -0, E1 0, E2 0, E3 0, E4 0} C_DIS
LIN {X 736.126, Y -394.037, Z 89.4, A 0, B 90, C -0, E1 0, E2 0, E3 0, E4 0} C_DIS
LIN {X 737.846, Y -400.523, Z 89.4, A 0, B 90, C -0, E1 0, E2 0, E3 0, E4 0} C_DIS
LIN {X 737.806, Y -401.841, Z 89.4, A 0, B 90, C -0, E1 0, E2 0, E3 0, E4 0} C_DIS
LIN {X 736.948, Y -402.848, Z 89.4, A 0, B 90, C -0, E1 0, E2 0, E3 0, E4 0} C_DIS
LIN {X 731.622, Y -406.93, Z 89.4, A 0, B 90, C -0, E1 0, E2 0, E3 0, E4 0} C_DIS
LIN {X 730.912, Y -408.002, Z 89.4, A 0, B 90, C -0, E1 0, E2 0, E3 0, E4 0} C_DIS
LIN {X 731.61, Y -409.109, Z 89.4, A 0, B 90, C -0, E1 0, E2 0, E3 0, E4 0} C_DIS
LIN {X 736.342, Y -413.866, Z 89.4, A 0, B 90, C -0, E1 0, E2 0, E3 0, E4 0} C_DIS
LIN {X 736.967, Y -415.027, Z 89.4, A 0, B 90, C -0, E1 0, E2 0, E3 0, E4 0} C_DIS
LIN {X 736.727, Y -416.328, Z 89.4, A 0, B 90, C -0, E1 0, E2 0, E3 0, E4 0} C_DIS
LIN {X 734.156, Y -422.526, Z 89.4, A 0, B 90, C -0, E1 0, E2 0, E3 0, E4 0} C_DIS
LIN {X 734.077, Y -423.81, Z 89.4, A 0, B 90, C -0, E1 0, E2 0, E3 0, E4 0} C_DIS
LIN {X 735.235, Y -424.419, Z 89.4, A 0, B 90, C -0, E1 0, E2 0, E3 0, E4 0} C_DIS
LIN {X 741.711, Y -426.173, Z 89.4, A 0, B 90, C -0, E1 0, E2 0, E3 0, E4 0} C_DIS
LIN {X 742.833, Y -426.866, Z 89.4, A 0, B 90, C -0, E1 0, E2 0, E3 0, E4 0} C_DIS
LIN {X 743.276, Y -428.113, Z 89.4, A 0, B 90, C -0, E1 0, E2 0, E3 0, E4 0} C_DIS
LIN {X 744.148, Y -434.766, Z 89.4, A 0, B 90, C -0, E1 0, E2 0, E3 0, E4 0} C_DIS
LIN {X 744.722, Y -435.918, Z 89.4, A 0, B 90, C -0, E1 0, E2 0, E3 0, E4 0} C_DIS
LIN {X 746.029, Y -435.866, Z 89.4, A 0, B 90, C -0, E1 0, E2 0, E3 0, E4 0} C_DIS
LIN {X 752.515, Y -434.147, Z 89.4, A 0, B 90, C -0, E1 0, E2 0, E3 0, E4 0} C_DIS
LIN {X 753.833, Y -434.186, Z 89.4, A 0, B 90, C -0, E1 0, E2 0, E3 0, E4 0} C_DIS
LIN {X 754.84, Y -435.045, Z 89.4, A 0, B 90, C -0, E1 0, E2 0, E3 0, E4 0} C_DIS
LIN {X 758.922, Y -440.37, Z 89.4, A 0, B 90, C -0, E1 0, E2 0, E3 0, E4 0} C_DIS
LIN {X 759.994, Y -441.081, Z 89.4, A 0, B 90, C -0, E1 0, E2 0, E3 0, E4 0} C_DIS
LIN {X 761.101, Y -440.383, Z 89.4, A 0, B 90, C -0, E1 0, E2 0, E3 0, E4 0} C_DIS
LIN {X 765.858, Y -435.651, Z 89.4, A 0, B 90, C -0, E1 0, E2 0, E3 0, E4 0} C_DIS
LIN {X 767.019, Y -435.026, Z 89.4, A 0, B 90, C -0, E1 0, E2 0, E3 0, E4 0} C_DIS
LIN {X 768.321, Y -435.265, Z 89.4, A 0, B 90, C -0, E1 0, E2 0, E3 0, E4 0} C_DIS
LIN {X 774.518, Y -437.837, Z 89.4, A 0, B 90, C -0, E1 0, E2 0, E3 0, E4 0} C_DIS
LIN {X 775.802, Y -437.916, Z 89.4, A 0, B 90, C -0, E1 0, E2 0, E3 0, E4 0} C_DIS
LIN {X 776.412, Y -436.758, Z 89.4, A 0, B 90, C -0, E1 0, E2 0, E3 0, E4 0} C_DIS
LIN {X 778.166, Y -430.281, Z 89.4, A 0, B 90, C -0, E1 0, E2 0, E3 0, E4 0} C_DIS
LIN {X 778.859, Y -429.16, Z 89.4, A 0, B 90, C -0, E1 0, E2 0, E3 0, E4 0} C_DIS
LIN {X 780.106, Y -428.716, Z 89.4, A 0, B 90, C -0, E1 0, E2 0, E3 0, E4 0} C_DIS
LIN {X 786.759, Y -427.844, Z 89.4, A 0, B 90, C -0, E1 0, E2 0, E3 0, E4 0} C_DIS
LIN {X 787.91, Y -427.271, Z 89.4, A 0, B 90, C -0, E1 0, E2 0, E3 0, E4 0} C_DIS
LIN {X 787.859, Y -425.963, Z 89.4, A 0, B 90, C -0, E1 0, E2 0, E3 0, E4 0} C_DIS
LIN {X 786.139, Y -419.477, Z 89.4, A 0, B 90, C -0, E1 0, E2 0, E3 0, E4 0} C_DIS
LIN {X 786.179, Y -418.159, Z 89.4, A 0, B 90, C -0, E1 0, E2 0, E3 0, E4 0} C_DIS
LIN {X 787.037, Y -417.152, Z 89.4, A 0, B 90, C -0, E1 0, E2 0, E3 0, E4 0} C_DIS
LIN {X 792.363, Y -413.07, Z 89.4, A 0, B 90, C -0, E1 0, E2 0, E3 0, E4 0} C_DIS
LIN {X 793.073, Y -411.998, Z 89.4, A 0, B 90, C -0, E1 0, E2 0, E3 0, E4 0} C_DIS
LIN {X 792.375, Y -410.891, Z 89.4, A 0, B 90, C -0, E1 0, E2 0, E3 0, E4 0} C_DIS
LIN {X 787.643, Y -406.134, Z 89.4, A 0, B 90, C -0, E1 0, E2 0, E3 0, E4 0} C_DIS
LIN {X 787.018, Y -404.973, Z 89.4, A 0, B 90, C -0, E1 0, E2 0, E3 0, E4 0} C_DIS
LIN {X 787.258, Y -403.672, Z 89.4, A 0, B 90, C -0, E1 0, E2 0, E3 0, E4 0} C_DIS
LIN {X 789.829, Y -397.474, Z 89.4, A 0, B 90, C -0, E1 0, E2 0, E3 0, E4 0} C_DIS
LIN {X 789.908, Y -396.19, Z 89.4, A 0, B 90, C -0, E1 0, E2 0, E3 0, E4 0} C_DIS
LIN {X 788.75, Y -395.581, Z 89.4, A 0, B 90, C -0, E1 0, E2 0, E3 0, E4 0} C_DIS
LIN {X 782.274, Y -393.827, Z 89.4, A 0, B 90, C -0, E1 0, E2 0, E3 0, E4 0} C_DIS
LIN {X 781.152, Y -393.134, Z 89.4, A 0, B 90, C -0, E1 0, E2 0, E3 0, E4 0} C_DIS
LIN {X 780.709, Y -391.887, Z 89.4, A 0, B 90, C -0, E1 0, E2 0, E3 0, E4 0} C_DIS
LIN {X 779.837, Y -385.234, Z 89.4, A 0, B 90, C -0, E1 0, E2 0, E3 0, E4 0} C_DIS
LIN {X 779.263, Y -384.082, Z 89.4, A 0, B 90, C -0, E1 0, E2 0, E3 0, E4 0} C_DIS
LIN {X 777.956, Y -384.134, Z 89.4, A 0, B 90, C -0, E1 0, E2 0, E3 0, E4 0} C_DIS
LIN {X 772.767, Y -385.509, Z 89.4, A 0, B 90, C -0, E1 0, E2 0, E3 0, E4 0} C_DIS
LIN {X 771.215, Y -385.902, Z 90.05, A 0, B 90, C -0, E1 0, E2 0, E3 0, E4 0} C_DIS
LIN {X 769.904, Y -385.874, Z 90.05, A 0, B 90, C -0, E1 0, E2 0, E3 0, E4 0} C_DIS
LIN {X 768.895, Y -385.029, Z 90.05, A 0, B 90, C -0, E1 0, E2 0, E3 0, E4 0} C_DIS
LIN {X 764.79, Y -379.767, Z 90.05, A 0, B 90, C -0, E1 0, E2 0, E3 0, E4 0} C_DIS
LIN {X 763.717, Y -379.069, Z 90.05, A 0, B 90, C -0, E1 0, E2 0, E3 0, E4 0} C_DIS
LIN {X 762.622, Y -379.773, Z 90.05, A 0, B 90, C -0, E1 0, E2 0, E3 0, E4 0} C_DIS
LIN {X 757.931, Y -384.52, Z 90.05, A 0, B 90, C -0, E1 0, E2 0, E3 0, E4 0} C_DIS
LIN {X 756.781, Y -385.151, Z 90.05, A 0, B 90, C -0, E1 0, E2 0, E3 0, E4 0} C_DIS
LIN {X 755.485, Y -384.924, Z 90.05, A 0, B 90, C -0, E1 0, E2 0, E3 0, E4 0} C_DIS
LIN {X 749.298, Y -382.419, Z 90.05, A 0, B 90, C -0, E1 0, E2 0, E3 0, E4 0} C_DIS
LIN {X 748.021, Y -382.351, Z 90.05, A 0, B 90, C -0, E1 0, E2 0, E3 0, E4 0} C_DIS
LIN {X 747.424, Y -383.508, Z 90.05, A 0, B 90, C -0, E1 0, E2 0, E3 0, E4 0} C_DIS
LIN {X 745.735, Y -389.964, Z 90.05, A 0, B 90, C -0, E1 0, E2 0, E3 0, E4 0} C_DIS
LIN {X 745.055, Y -391.086, Z 90.05, A 0, B 90, C -0, E1 0, E2 0, E3 0, E4 0} C_DIS
LIN {X 743.818, Y -391.537, Z 90.05, A 0, B 90, C -0, E1 0, E2 0, E3 0, E4 0} C_DIS
LIN {X 737.208, Y -392.461, Z 90.05, A 0, B 90, C -0, E1 0, E2 0, E3 0, E4 0} C_DIS
LIN {X 736.068, Y -393.041, Z 90.05, A 0, B 90, C -0, E1 0, E2 0, E3 0, E4 0} C_DIS
LIN {X 736.13, Y -394.341, Z 90.05, A 0, B 90, C -0, E1 0, E2 0, E3 0, E4 0} C_DIS
LIN {X 737.895, Y -400.777, Z 90.05, A 0, B 90, C -0, E1 0, E2 0, E3 0, E4 0} C_DIS
LIN {X 737.867, Y -402.089, Z 90.05, A 0, B 90, C -0, E1 0, E2 0, E3 0, E4 0} C_DIS
LIN {X 737.022, Y -403.098, Z 90.05, A 0, B 90, C -0, E1 0, E2 0, E3 0, E4 0} C_DIS
LIN {X 731.759, Y -407.203, Z 90.05, A 0, B 90, C -0, E1 0, E2 0, E3 0, E4 0} C_DIS
LIN {X 731.062, Y -408.275, Z 90.05, A 0, B 90, C -0, E1 0, E2 0, E3 0, E4 0} C_DIS
LIN {X 731.765, Y -409.37, Z 90.05, A 0, B 90, C -0, E1 0, E2 0, E3 0, E4 0} C_DIS
LIN {X 736.512, Y -414.062, Z 90.05, A 0, B 90, C -0, E1 0, E2 0, E3 0, E4 0} C_DIS
LIN {X 737.143, Y -415.211, Z 90.05, A 0, B 90, C -0, E1 0, E2 0, E3 0, E4 0} C_DIS
LIN {X 736.916, Y -416.508, Z 90.05, A 0, B 90, C -0, E1 0, E2 0, E3 0, E4 0} C_DIS
LIN {X 734.411, Y -422.694, Z 90.05, A 0, B 90, C -0, E1 0, E2 0, E3 0, E4 0} C_DIS
LIN {X 734.343, Y -423.972, Z 90.05, A 0, B 90, C -0, E1 0, E2 0, E3 0, E4 0} C_DIS
LIN {X 735.5, Y -424.568, Z 90.05, A 0, B 90, C -0, E1 0, E2 0, E3 0, E4 0} C_DIS
LIN {X 741.957, Y -426.258, Z 90.05, A 0, B 90, C -0, E1 0, E2 0, E3 0, E4 0} C_DIS
LIN {X 743.078, Y -426.938, Z 90.05, A 0, B 90, C -0, E1 0, E2 0, E3 0, E4 0} C_DIS
LIN {X 743.53, Y -428.174, Z 90.05, A 0, B 90, C -0, E1 0, E2 0, E3 0, E4 0} C_DIS
LIN {X 744.453, Y -434.784, Z 90.05, A 0, B 90, C -0, E1 0, E2 0, E3 0, E4 0} C_DIS
LIN {X 745.033, Y -435.925, Z 90.05, A 0, B 90, C -0, E1 0, E2 0, E3 0, E4 0} C_DIS
LIN {X 746.333, Y -435.863, Z 90.05, A 0, B 90, C -0, E1 0, E2 0, E3 0, E4 0} C_DIS
LIN {X 752.77, Y -434.098, Z 90.05, A 0, B 90, C -0, E1 0, E2 0, E3 0, E4 0} C_DIS
LIN {X 754.081, Y -434.126, Z 90.05, A 0, B 90, C -0, E1 0, E2 0, E3 0, E4 0} C_DIS
LIN {X 755.09, Y -434.971, Z 90.05, A 0, B 90, C -0, E1 0, E2 0, E3 0, E4 0} C_DIS
LIN {X 759.195, Y -440.233, Z 90.05, A 0, B 90, C -0, E1 0, E2 0, E3 0, E4 0} C_DIS
LIN {X 760.268, Y -440.931, Z 90.05, A 0, B 90, C -0, E1 0, E2 0, E3 0, E4 0} C_DIS
LIN {X 761.363, Y -440.227, Z 90.05, A 0, B 90, C -0, E1 0, E2 0, E3 0, E4 0} C_DIS
LIN {X 766.054, Y -435.48, Z 90.05, A 0, B 90, C -0, E1 0, E2 0, E3 0, E4 0} C_DIS
LIN {X 767.204, Y -434.849, Z 90.05, A 0, B 90, C -0, E1 0, E2 0, E3 0, E4 0} C_DIS
LIN {X 768.5, Y -435.076, Z 90.05, A 0, B 90, C -0, E1 0, E2 0, E3 0, E4 0} C_DIS
LIN {X 774.686, Y -437.581, Z 90.05, A 0, B 90, C -0, E1 0, E2 0, E3 0, E4 0} C_DIS
LIN {X 775.964, Y -437.649, Z 90.05, A 0, B 90, C -0, E1 0, E2 0, E3 0, E4 0} C_DIS
LIN {X 776.561, Y -436.492, Z 90.05, A 0, B 90, C -0, E1 0, E2 0, E3 0, E4 0} C_DIS
LIN {X 778.25, Y -430.036, Z 90.05, A 0, B 90, C -0, E1 0, E2 0, E3 0, E4 0} C_DIS
LIN {X 778.93, Y -428.914, Z 90.05, A 0, B 90, C -0, E1 0, E2 0, E3 0, E4 0} C_DIS
LIN {X 780.167, Y -428.463, Z 90.05, A 0, B 90, C -0, E1 0, E2 0, E3 0, E4 0} C_DIS
LIN {X 786.777, Y -427.539, Z 90.05, A 0, B 90, C -0, E1 0, E2 0, E3 0, E4 0} C_DIS
LIN {X 787.917, Y -426.959, Z 90.05, A 0, B 90, C -0, E1 0, E2 0, E3 0, E4 0} C_DIS
LIN {X 787.855, Y -425.659, Z 90.05, A 0, B 90, C -0, E1 0, E2 0, E3 0, E4 0} C_DIS
LIN {X 786.09, Y -419.223, Z 90.05, A 0, B 90, C -0, E1 0, E2 0, E3 0, E4 0} C_DIS
LIN {X 786.118, Y -417.911, Z 90.05, A 0, B 90, C -0, E1 0, E2 0, E3 0, E4 0} C_DIS
LIN {X 786.963, Y -416.902, Z 90.05, A 0, B 90, C -0, E1 0, E2 0, E3 0, E4 0} C_DIS
LIN {X 792.226, Y -412.797, Z 90.05, A 0, B 90, C -0, E1 0, E2 0, E3 0, E4 0} C_DIS
LIN {X 792.923, Y -411.725, Z 90.05, A 0, B 90, C -0, E1 0, E2 0, E3 0, E4 0} C_DIS
LIN {X 792.22, Y -410.63, Z 90.05, A 0, B 90, C -0, E1 0, E2 0, E3 0, E4 0} C_DIS
LIN {X 787.473, Y -405.938, Z 90.05, A 0, B 90, C -0, E1 0, E2 0, E3 0, E4 0} C_DIS
LIN {X 786.842, Y -404.789, Z 90.05, A 0, B 90, C -0, E1 0, E2 0, E3 0, E4 0} C_DIS
LIN {X 787.069, Y -403.492, Z 90.05, A 0, B 90, C -0, E1 0, E2 0, E3 0, E4 0} C_DIS
LIN {X 789.574, Y -397.306, Z 90.05, A 0, B 90, C -0, E1 0, E2 0, E3 0, E4 0} C_DIS
LIN {X 789.642, Y -396.028, Z 90.05, A 0, B 90, C -0, E1 0, E2 0, E3 0, E4 0} C_DIS
LIN {X 788.485, Y -395.432, Z 90.05, A 0, B 90, C -0, E1 0, E2 0, E3 0, E4 0} C_DIS
LIN {X 782.028, Y -393.742, Z 90.05, A 0, B 90, C -0, E1 0, E2 0, E3 0, E4 0} C_DIS
LIN {X 780.907, Y -393.062, Z 90.05, A 0, B 90, C -0, E1 0, E2 0, E3 0, E4 0} C_DIS
LIN {X 780.455, Y -391.826, Z 90.05, A 0, B 90, C -0, E1 0, E2 0, E3 0, E4 0} C_DIS
LIN {X 779.532, Y -385.216, Z 90.05, A 0, B 90, C -0, E1 0, E2 0, E3 0, E4 0} C_DIS
LIN {X 778.952, Y -384.075, Z 90.05, A 0, B 90, C -0, E1 0, E2 0, E3 0, E4 0} C_DIS
LIN {X 777.651, Y -384.137, Z 90.05, A 0, B 90, C -0, E1 0, E2 0, E3 0, E4 0} C_DIS
LIN {X 772.502, Y -385.549, Z 90.05, A 0, B 90, C -0, E1 0, E2 0, E3 0, E4 0} C_DIS
LIN {X 770.963, Y -385.953, Z 90.7, A 0, B 90, C -0, E1 0, E2 0, E3 0, E4 0} C_DIS
LIN {X 769.658, Y -385.936, Z 90.7, A 0, B 90, C -0, E1 0, E2 0, E3 0, E4 0} C_DIS
LIN {X 768.648, Y -385.104, Z 90.7, A 0, B 90, C -0, E1 0, E2 0, E3 0, E4 0} C_DIS
LIN {X 764.52, Y -379.904, Z 90.7, A 0, B 90, C -0, E1 0, E2 0, E3 0, E4 0} C_DIS
LIN {X 763.447, Y -379.219, Z 90.7, A 0, B 90, C -0, E1 0, E2 0, E3 0, E4 0} C_DIS
LIN {X 762.364, Y -379.928, Z 90.7, A 0, B 90, C -0, E1 0, E2 0, E3 0, E4 0} C_DIS
LIN {X 757.738, Y -384.689, Z 90.7, A 0, B 90, C -0, E1 0, E2 0, E3 0, E4 0} C_DIS
LIN {X 756.599, Y -385.327, Z 90.7, A 0, B 90, C -0, E1 0, E2 0, E3 0, E4 0} C_DIS
LIN {X 755.308, Y -385.112, Z 90.7, A 0, B 90, C -0, E1 0, E2 0, E3 0, E4 0} C_DIS
LIN {X 749.133, Y -382.672, Z 90.7, A 0, B 90, C -0, E1 0, E2 0, E3 0, E4 0} C_DIS
LIN {X 747.862, Y -382.615, Z 90.7, A 0, B 90, C -0, E1 0, E2 0, E3 0, E4 0} C_DIS
LIN {X 747.278, Y -383.771, Z 90.7, A 0, B 90, C -0, E1 0, E2 0, E3 0, E4 0} C_DIS
LIN {X 745.652, Y -390.208, Z 90.7, A 0, B 90, C -0, E1 0, E2 0, E3 0, E4 0} C_DIS
LIN {X 744.985, Y -391.329, Z 90.7, A 0, B 90, C -0, E1 0, E2 0, E3 0, E4 0} C_DIS
LIN {X 743.759, Y -391.788, Z 90.7, A 0, B 90, C -0, E1 0, E2 0, E3 0, E4 0} C_DIS
LIN {X 737.192, Y -392.763, Z 90.7, A 0, B 90, C -0, E1 0, E2 0, E3 0, E4 0} C_DIS
LIN {X 736.063, Y -393.35, Z 90.7, A 0, B 90, C -0, E1 0, E2 0, E3 0, E4 0} C_DIS
LIN {X 736.135, Y -394.642, Z 90.7, A 0, B 90, C -0, E1 0, E2 0, E3 0, E4 0} C_DIS
LIN {X 737.945, Y -401.03, Z 90.7, A 0, B 90, C -0, E1 0, E2 0, E3 0, E4 0} C_DIS
LIN {X 737.928, Y -402.334, Z 90.7, A 0, B 90, C -0, E1 0, E2 0, E3 0, E4 0} C_DIS
LIN {X 737.096, Y -403.345, Z 90.7, A 0, B 90, C -0, E1 0, E2 0, E3 0, E4 0} C_DIS
LIN {X 731.896, Y -407.472, Z 90.7, A 0, B 90, C -0, E1 0, E2 0, E3 0, E4 0} C_DIS
LIN {X 731.211, Y -408.545, Z 90.7, A 0, B 90, C -0, E1 0, E2 0, E3 0, E4 0} C_DIS
LIN {X 731.921, Y -409.628, Z 90.7, A 0, B 90, C -0, E1 0, E2 0, E3 0, E4 0} C_DIS
LIN {X 736.682, Y -414.255, Z 90.7, A 0, B 90, C -0, E1 0, E2 0, E3 0, E4 0} C_DIS
LIN {X 737.319, Y -415.393, Z 90.7, A 0, B 90, C -0, E1 0, E2 0, E3 0, E4 0} C_DIS
LIN {X 737.104, Y -416.685, Z 90.7, A 0, B 90, C -0, E1 0, E2 0, E3 0, E4 0} C_DIS
LIN {X 734.665, Y -422.859, Z 90.7, A 0, B 90, C -0, E1 0, E2 0, E3 0, E4 0} C_DIS
LIN {X 734.608, Y -424.131, Z 90.7, A 0, B 90, C -0, E1 0, E2 0, E3 0, E4 0} C_DIS
LIN {X 735.764, Y -424.714, Z 90.7, A 0, B 90, C -0, E1 0, E2 0, E3 0, E4 0} C_DIS
LIN {X 742.2, Y -426.34, Z 90.7, A 0, B 90, C -0, E1 0, E2 0, E3 0, E4 0} C_DIS
LIN {X 743.322, Y -427.007, Z 90.7, A 0, B 90, C -0, E1 0, E2 0, E3 0, E4 0} C_DIS
LIN {X 743.781, Y -428.233, Z 90.7, A 0, B 90, C -0, E1 0, E2 0, E3 0, E4 0} C_DIS
LIN {X 744.755, Y -434.8, Z 90.7, A 0, B 90, C -0, E1 0, E2 0, E3 0, E4 0} C_DIS
LIN {X 745.342, Y -435.93, Z 90.7, A 0, B 90, C -0, E1 0, E2 0, E3 0, E4 0} C_DIS
LIN {X 746.635, Y -435.857, Z 90.7, A 0, B 90, C -0, E1 0, E2 0, E3 0, E4 0} C_DIS
LIN {X 753.022, Y -434.047, Z 90.7, A 0, B 90, C -0, E1 0, E2 0, E3 0, E4 0} C_DIS
LIN {X 754.327, Y -434.064, Z 90.7, A 0, B 90, C -0, E1 0, E2 0, E3 0, E4 0} C_DIS
LIN {X 755.337, Y -434.896, Z 90.7, A 0, B 90, C -0, E1 0, E2 0, E3 0, E4 0} C_DIS
LIN {X 759.465, Y -440.096, Z 90.7, A 0, B 90, C -0, E1 0, E2 0, E3 0, E4 0} C_DIS
LIN {X 760.538, Y -440.781, Z 90.7, A 0, B 90, C -0, E1 0, E2 0, E3 0, E4 0} C_DIS
LIN {X 761.621, Y -440.072, Z 90.7, A 0, B 90, C -0, E1 0, E2 0, E3 0, E4 0} C_DIS
LIN {X 766.247, Y -435.311, Z 90.7, A 0, B 90, C -0, E1 0, E2 0, E3 0, E4 0} C_DIS
LIN {X 767.386, Y -434.673, Z 90.7, A 0, B 90, C -0, E1 0, E2 0, E3 0, E4 0} C_DIS
LIN {X 768.677, Y -434.888, Z 90.7, A 0, B 90, C -0, E1 0, E2 0, E3 0, E4 0} C_DIS
LIN {X 774.852, Y -437.328, Z 90.7, A 0, B 90, C -0, E1 0, E2 0, E3 0, E4 0} C_DIS
LIN {X 776.123, Y -437.385, Z 90.7, A 0, B 90, C -0, E1 0, E2 0, E3 0, E4 0} C_DIS
LIN {X 776.706, Y -436.229, Z 90.7, A 0, B 90, C -0, E1 0, E2 0, E3 0, E4 0} C_DIS
LIN {X 778.333, Y -429.792, Z 90.7, A 0, B 90, C -0, E1 0, E2 0, E3 0, E4 0} C_DIS
LIN {X 779, Y -428.671, Z 90.7, A 0, B 90, C -0, E1 0, E2 0, E3 0, E4 0} C_DIS
LIN {X 780.226, Y -428.212, Z 90.7, A 0, B 90, C -0, E1 0, E2 0, E3 0, E4 0} C_DIS
LIN {X 786.793, Y -427.237, Z 90.7, A 0, B 90, C -0, E1 0, E2 0, E3 0, E4 0} C_DIS
LIN {X 787.922, Y -426.65, Z 90.7, A 0, B 90, C -0, E1 0, E2 0, E3 0, E4 0} C_DIS
LIN {X 787.85, Y -425.358, Z 90.7, A 0, B 90, C -0, E1 0, E2 0, E3 0, E4 0} C_DIS
LIN {X 786.04, Y -418.97, Z 90.7, A 0, B 90, C -0, E1 0, E2 0, E3 0, E4 0} C_DIS
LIN {X 786.057, Y -417.666, Z 90.7, A 0, B 90, C -0, E1 0, E2 0, E3 0, E4 0} C_DIS
LIN {X 786.889, Y -416.655, Z 90.7, A 0, B 90, C -0, E1 0, E2 0, E3 0, E4 0} C_DIS
LIN {X 792.089, Y -412.528, Z 90.7, A 0, B 90, C -0, E1 0, E2 0, E3 0, E4 0} C_DIS
LIN {X 792.774, Y -411.455, Z 90.7, A 0, B 90, C -0, E1 0, E2 0, E3 0, E4 0} C_DIS
LIN {X 792.064, Y -410.372, Z 90.7, A 0, B 90, C -0, E1 0, E2 0, E3 0, E4 0} C_DIS
LIN {X 787.303, Y -405.745, Z 90.7, A 0, B 90, C -0, E1 0, E2 0, E3 0, E4 0} C_DIS
LIN {X 786.666, Y -404.607, Z 90.7, A 0, B 90, C -0, E1 0, E2 0, E3 0, E4 0} C_DIS
LIN {X 786.881, Y -403.315, Z 90.7, A 0, B 90, C -0, E1 0, E2 0, E3 0, E4 0} C_DIS
LIN {X 789.32, Y -397.141, Z 90.7, A 0, B 90, C -0, E1 0, E2 0, E3 0, E4 0} C_DIS
LIN {X 789.377, Y -395.869, Z 90.7, A 0, B 90, C -0, E1 0, E2 0, E3 0, E4 0} C_DIS
LIN {X 788.221, Y -395.286, Z 90.7, A 0, B 90, C -0, E1 0, E2 0, E3 0, E4 0} C_DIS
LIN {X 781.785, Y -393.66, Z 90.7, A 0, B 90, C -0, E1 0, E2 0, E3 0, E4 0} C_DIS
LIN {X 780.663, Y -392.993, Z 90.7, A 0, B 90, C -0, E1 0, E2 0, E3 0, E4 0} C_DIS
LIN {X 780.204, Y -391.767, Z 90.7, A 0, B 90, C -0, E1 0, E2 0, E3 0, E4 0} C_DIS
LIN {X 779.23, Y -385.2, Z 90.7, A 0, B 90, C -0, E1 0, E2 0, E3 0, E4 0} C_DIS
LIN {X 778.643, Y -384.07, Z 90.7, A 0, B 90, C -0, E1 0, E2 0, E3 0, E4 0} C_DIS
LIN {X 777.35, Y -384.143, Z 90.7, A 0, B 90, C -0, E1 0, E2 0, E3 0, E4 0} C_DIS
LIN {X 772.24, Y -385.591, Z 90.7, A 0, B 90, C -0, E1 0, E2 0, E3 0, E4 0} C_DIS
LIN {X 770.714, Y -386.004, Z 91.35, A 0, B 90, C -0, E1 0, E2 0, E3 0, E4 0} C_DIS
LIN {X 769.416, Y -385.998, Z 91.35, A 0, B 90, C -0, E1 0, E2 0, E3 0, E4 0} C_DIS
LIN {X 768.403, Y -385.179, Z 91.35, A 0, B 90, C -0, E1 0, E2 0, E3 0, E4 0} C_DIS
LIN {X 764.254, Y -380.041, Z 91.35, A 0, B 90, C -0, E1 0, E2 0, E3 0, E4 0} C_DIS
LIN {X 763.181, Y -379.369, Z 91.35, A 0, B 90, C -0, E1 0, E2 0, E3 0, E4 0} C_DIS
LIN {X 762.109, Y -380.084, Z 91.35, A 0, B 90, C -0, E1 0, E2 0, E3 0, E4 0} C_DIS
LIN {X 757.547, Y -384.858, Z 91.35, A 0, B 90, C -0, E1 0, E2 0, E3 0, E4 0} C_DIS
LIN {X 756.42, Y -385.502, Z 91.35, A 0, B 90, C -0, E1 0, E2 0, E3 0, E4 0} C_DIS
LIN {X 755.134, Y -385.299, Z 91.35, A 0, B 90, C -0, E1 0, E2 0, E3 0, E4 0} C_DIS
LIN {X 748.971, Y -382.924, Z 91.35, A 0, B 90, C -0, E1 0, E2 0, E3 0, E4 0} C_DIS
LIN {X 747.706, Y -382.878, Z 91.35, A 0, B 90, C -0, E1 0, E2 0, E3 0, E4 0} C_DIS
LIN {X 747.135, Y -384.033, Z 91.35, A 0, B 90, C -0, E1 0, E2 0, E3 0, E4 0} C_DIS
LIN {X 745.572, Y -390.449, Z 91.35, A 0, B 90, C -0, E1 0, E2 0, E3 0, E4 0} C_DIS
LIN {X 744.918, Y -391.57, Z 91.35, A 0, B 90, C -0, E1 0, E2 0, E3 0, E4 0} C_DIS
LIN {X 743.702, Y -392.038, Z 91.35, A 0, B 90, C -0, E1 0, E2 0, E3 0, E4 0} C_DIS
LIN {X 737.178, Y -393.062, Z 91.35, A 0, B 90, C -0, E1 0, E2 0, E3 0, E4 0} C_DIS
LIN {X 736.059, Y -393.655, Z 91.35, A 0, B 90, C -0, E1 0, E2 0, E3 0, E4 0} C_DIS
LIN {X 736.143, Y -394.94, Z 91.35, A 0, B 90, C -0, E1 0, E2 0, E3 0, E4 0} C_DIS
LIN {X 737.997, Y -401.279, Z 91.35, A 0, B 90, C -0, E1 0, E2 0, E3 0, E4 0} C_DIS
LIN {X 737.991, Y -402.577, Z 91.35, A 0, B 90, C -0, E1 0, E2 0, E3 0, E4 0} C_DIS
LIN {X 737.171, Y -403.589, Z 91.35, A 0, B 90, C -0, E1 0, E2 0, E3 0, E4 0} C_DIS
LIN {X 732.034, Y -407.739, Z 91.35, A 0, B 90, C -0, E1 0, E2 0, E3 0, E4 0} C_DIS
LIN {X 731.361, Y -408.812, Z 91.35, A 0, B 90, C -0, E1 0, E2 0, E3 0, E4 0} C_DIS
LIN {X 732.076, Y -409.883, Z 91.35, A 0, B 90, C -0, E1 0, E2 0, E3 0, E4 0} C_DIS
LIN {X 736.851, Y -414.445, Z 91.35, A 0, B 90, C -0, E1 0, E2 0, E3 0, E4 0} C_DIS
LIN {X 737.495, Y -415.572, Z 91.35, A 0, B 90, C -0, E1 0, E2 0, E3 0, E4 0} C_DIS
LIN {X 737.292, Y -416.859, Z 91.35, A 0, B 90, C -0, E1 0, E2 0, E3 0, E4 0} C_DIS
LIN {X 734.917, Y -423.021, Z 91.35, A 0, B 90, C -0, E1 0, E2 0, E3 0, E4 0} C_DIS
LIN {X 734.871, Y -424.286, Z 91.35, A 0, B 90, C -0, E1 0, E2 0, E3 0, E4 0} C_DIS
LIN {X 736.026, Y -424.857, Z 91.35, A 0, B 90, C -0, E1 0, E2 0, E3 0, E4 0} C_DIS
LIN {X 742.442, Y -426.421, Z 91.35, A 0, B 90, C -0, E1 0, E2 0, E3 0, E4 0} C_DIS
LIN {X 743.563, Y -427.075, Z 91.35, A 0, B 90, C -0, E1 0, E2 0, E3 0, E4 0} C_DIS
LIN {X 744.03, Y -428.29, Z 91.35, A 0, B 90, C -0, E1 0, E2 0, E3 0, E4 0} C_DIS
LIN {X 745.055, Y -434.814, Z 91.35, A 0, B 90, C -0, E1 0, E2 0, E3 0, E4 0} C_DIS
LIN {X 745.648, Y -435.933, Z 91.35, A 0, B 90, C -0, E1 0, E2 0, E3 0, E4 0} C_DIS
LIN {X 746.933, Y -435.85, Z 91.35, A 0, B 90, C -0, E1 0, E2 0, E3 0, E4 0} C_DIS
LIN {X 753.271, Y -433.996, Z 91.35, A 0, B 90, C -0, E1 0, E2 0, E3 0, E4 0} C_DIS
LIN {X 754.569, Y -434.002, Z 91.35, A 0, B 90, C -0, E1 0, E2 0, E3 0, E4 0} C_DIS
LIN {X 755.582, Y -434.821, Z 91.35, A 0, B 90, C -0, E1 0, E2 0, E3 0, E4 0} C_DIS
LIN {X 759.731, Y -439.959, Z 91.35, A 0, B 90, C -0, E1 0, E2 0, E3 0, E4 0} C_DIS
LIN {X 760.804, Y -440.631, Z 91.35, A 0, B 90, C -0, E1 0, E2 0, E3 0, E4 0} C_DIS
LIN {X 761.876, Y -439.916, Z 91.35, A 0, B 90, C -0, E1 0, E2 0, E3 0, E4 0} C_DIS
LIN {X 766.438, Y -435.142, Z 91.35, A 0, B 90, C -0, E1 0, E2 0, E3 0, E4 0} C_DIS
LIN {X 767.565, Y -434.498, Z 91.35, A 0, B 90, C -0, E1 0, E2 0, E3 0, E4 0} C_DIS
LIN {X 768.851, Y -434.701, Z 91.35, A 0, B 90, C -0, E1 0, E2 0, E3 0, E4 0} C_DIS
LIN {X 775.013, Y -437.076, Z 91.35, A 0, B 90, C -0, E1 0, E2 0, E3 0, E4 0} C_DIS
LIN {X 776.279, Y -437.122, Z 91.35, A 0, B 90, C -0, E1 0, E2 0, E3 0, E4 0} C_DIS
LIN {X 776.849, Y -435.967, Z 91.35, A 0, B 90, C -0, E1 0, E2 0, E3 0, E4 0} C_DIS
LIN {X 778.413, Y -429.551, Z 91.35, A 0, B 90, C -0, E1 0, E2 0, E3 0, E4 0} C_DIS
LIN {X 779.067, Y -428.43, Z 91.35, A 0, B 90, C -0, E1 0, E2 0, E3 0, E4 0} C_DIS
LIN {X 780.283, Y -427.962, Z 91.35, A 0, B 90, C -0, E1 0, E2 0, E3 0, E4 0} C_DIS
LIN {X 786.807, Y -426.938, Z 91.35, A 0, B 90, C -0, E1 0, E2 0, E3 0, E4 0} C_DIS
LIN {X 787.926, Y -426.345, Z 91.35, A 0, B 90, C -0, E1 0, E2 0, E3 0, E4 0} C_DIS
LIN {X 787.842, Y -425.06, Z 91.35, A 0, B 90, C -0, E1 0, E2 0, E3 0, E4 0} C_DIS
LIN {X 785.988, Y -418.721, Z 91.35, A 0, B 90, C -0, E1 0, E2 0, E3 0, E4 0} C_DIS
LIN {X 785.994, Y -417.423, Z 91.35, A 0, B 90, C -0, E1 0, E2 0, E3 0, E4 0} C_DIS
LIN {X 786.813, Y -416.411, Z 91.35, A 0, B 90, C -0, E1 0, E2 0, E3 0, E4 0} C_DIS
LIN {X 791.951, Y -412.261, Z 91.35, A 0, B 90, C -0, E1 0, E2 0, E3 0, E4 0} C_DIS
LIN {X 792.624, Y -411.188, Z 91.35, A 0, B 90, C -0, E1 0, E2 0, E3 0, E4 0} C_DIS
LIN {X 791.909, Y -410.117, Z 91.35, A 0, B 90, C -0, E1 0, E2 0, E3 0, E4 0} C_DIS
LIN {X 787.134, Y -405.555, Z 91.35, A 0, B 90, C -0, E1 0, E2 0, E3 0, E4 0} C_DIS
LIN {X 786.49, Y -404.428, Z 91.35, A 0, B 90, C -0, E1 0, E2 0, E3 0, E4 0} C_DIS
LIN {X 786.693, Y -403.141, Z 91.35, A 0, B 90, C -0, E1 0, E2 0, E3 0, E4 0} C_DIS
LIN {X 789.068, Y -396.979, Z 91.35, A 0, B 90, C -0, E1 0, E2 0, E3 0, E4 0} C_DIS
LIN {X 789.114, Y -395.714, Z 91.35, A 0, B 90, C -0, E1 0, E2 0, E3 0, E4 0} C_DIS
LIN {X 787.959, Y -395.143, Z 91.35, A 0, B 90, C -0, E1 0, E2 0, E3 0, E4 0} C_DIS
LIN {X 781.543, Y -393.579, Z 91.35, A 0, B 90, C -0, E1 0, E2 0, E3 0, E4 0} C_DIS
LIN {X 780.422, Y -392.925, Z 91.35, A 0, B 90, C -0, E1 0, E2 0, E3 0, E4 0} C_DIS
LIN {X 779.955, Y -391.71, Z 91.35, A 0, B 90, C -0, E1 0, E2 0, E3 0, E4 0} C_DIS
LIN {X 778.93, Y -385.186, Z 91.35, A 0, B 90, C -0, E1 0, E2 0, E3 0, E4 0} C_DIS
LIN {X 778.337, Y -384.067, Z 91.35, A 0, B 90, C -0, E1 0, E2 0, E3 0, E4 0} C_DIS
LIN {X 777.052, Y -384.15, Z 91.35, A 0, B 90, C -0, E1 0, E2 0, E3 0, E4 0} C_DIS
LIN {X 771.981, Y -385.633, Z 91.35, A 0, B 90, C -0, E1 0, E2 0, E3 0, E4 0} C_DIS
LIN {X 770.467, Y -386.056, Z 92, A 0, B 90, C -0, E1 0, E2 0, E3 0, E4 0} C_DIS
LIN {X 769.176, Y -386.061, Z 92, A 0, B 90, C -0, E1 0, E2 0, E3 0, E4 0} C_DIS
LIN {X 768.162, Y -385.255, Z 92, A 0, B 90, C -0, E1 0, E2 0, E3 0, E4 0} C_DIS
LIN {X 763.991, Y -380.179, Z 92, A 0, B 90, C -0, E1 0, E2 0, E3 0, E4 0} C_DIS
LIN {X 762.918, Y -379.519, Z 92, A 0, B 90, C -0, E1 0, E2 0, E3 0, E4 0} C_DIS
LIN {X 761.858, Y -380.239, Z 92, A 0, B 90, C -0, E1 0, E2 0, E3 0, E4 0} C_DIS
LIN {X 757.36, Y -385.027, Z 92, A 0, B 90, C -0, E1 0, E2 0, E3 0, E4 0} C_DIS
LIN {X 756.244, Y -385.677, Z 92, A 0, B 90, C -0, E1 0, E2 0, E3 0, E4 0} C_DIS
LIN {X 754.963, Y -385.485, Z 92, A 0, B 90, C -0, E1 0, E2 0, E3 0, E4 0} C_DIS
LIN {X 748.812, Y -383.175, Z 92, A 0, B 90, C -0, E1 0, E2 0, E3 0, E4 0} C_DIS
LIN {X 747.553, Y -383.14, Z 92, A 0, B 90, C -0, E1 0, E2 0, E3 0, E4 0} C_DIS
LIN {X 746.995, Y -384.293, Z 92, A 0, B 90, C -0, E1 0, E2 0, E3 0, E4 0} C_DIS
LIN {X 745.494, Y -390.689, Z 92, A 0, B 90, C -0, E1 0, E2 0, E3 0, E4 0} C_DIS
LIN {X 744.852, Y -391.81, Z 92, A 0, B 90, C -0, E1 0, E2 0, E3 0, E4 0} C_DIS
LIN {X 743.647, Y -392.285, Z 92, A 0, B 90, C -0, E1 0, E2 0, E3 0, E4 0} C_DIS
LIN {X 737.166, Y -393.359, Z 92, A 0, B 90, C -0, E1 0, E2 0, E3 0, E4 0} C_DIS
LIN {X 736.058, Y -393.958, Z 92, A 0, B 90, C -0, E1 0, E2 0, E3 0, E4 0} C_DIS
LIN {X 736.151, Y -395.236, Z 92, A 0, B 90, C -0, E1 0, E2 0, E3 0, E4 0} C_DIS
LIN {X 738.049, Y -401.526, Z 92, A 0, B 90, C -0, E1 0, E2 0, E3 0, E4 0} C_DIS
LIN {X 738.054, Y -402.817, Z 92, A 0, B 90, C -0, E1 0, E2 0, E3 0, E4 0} C_DIS
LIN {X 737.247, Y -403.831, Z 92, A 0, B 90, C -0, E1 0, E2 0, E3 0, E4 0} C_DIS
LIN {X 732.171, Y -408.002, Z 92, A 0, B 90, C -0, E1 0, E2 0, E3 0, E4 0} C_DIS
LIN {X 731.511, Y -409.075, Z 92, A 0, B 90, C -0, E1 0, E2 0, E3 0, E4 0} C_DIS
LIN {X 732.231, Y -410.134, Z 92, A 0, B 90, C -0, E1 0, E2 0, E3 0, E4 0} C_DIS
LIN {X 737.019, Y -414.633, Z 92, A 0, B 90, C -0, E1 0, E2 0, E3 0, E4 0} C_DIS
LIN {X 737.669, Y -415.749, Z 92, A 0, B 90, C -0, E1 0, E2 0, E3 0, E4 0} C_DIS
LIN {X 737.478, Y -417.03, Z 92, A 0, B 90, C -0, E1 0, E2 0, E3 0, E4 0} C_DIS
LIN {X 735.167, Y -423.18, Z 92, A 0, B 90, C -0, E1 0, E2 0, E3 0, E4 0} C_DIS
LIN {X 735.132, Y -424.439, Z 92, A 0, B 90, C -0, E1 0, E2 0, E3 0, E4 0} C_DIS
LIN {X 736.286, Y -424.997, Z 92, A 0, B 90, C -0, E1 0, E2 0, E3 0, E4 0} C_DIS
LIN {X 742.682, Y -426.499, Z 92, A 0, B 90, C -0, E1 0, E2 0, E3 0, E4 0} C_DIS
LIN {X 743.802, Y -427.14, Z 92, A 0, B 90, C -0, E1 0, E2 0, E3 0, E4 0} C_DIS
LIN {X 744.277, Y -428.345, Z 92, A 0, B 90, C -0, E1 0, E2 0, E3 0, E4 0} C_DIS
LIN {X 745.351, Y -434.827, Z 92, A 0, B 90, C -0, E1 0, E2 0, E3 0, E4 0} C_DIS
LIN {X 745.95, Y -435.935, Z 92, A 0, B 90, C -0, E1 0, E2 0, E3 0, E4 0} C_DIS
LIN {X 747.228, Y -435.841, Z 92, A 0, B 90, C -0, E1 0, E2 0, E3 0, E4 0} C_DIS
LIN {X 753.518, Y -433.944, Z 92, A 0, B 90, C -0, E1 0, E2 0, E3 0, E4 0} C_DIS
LIN {X 754.809, Y -433.939, Z 92, A 0, B 90, C -0, E1 0, E2 0, E3 0, E4 0} C_DIS
LIN {X 755.823, Y -434.745, Z 92, A 0, B 90, C -0, E1 0, E2 0, E3 0, E4 0} C_DIS
LIN {X 759.994, Y -439.821, Z 92, A 0, B 90, C -0, E1 0, E2 0, E3 0, E4 0} C_DIS
LIN {X 761.067, Y -440.481, Z 92, A 0, B 90, C -0, E1 0, E2 0, E3 0, E4 0} C_DIS
LIN {X 762.127, Y -439.761, Z 92, A 0, B 90, C -0, E1 0, E2 0, E3 0, E4 0} C_DIS
LIN {X 766.625, Y -434.973, Z 92, A 0, B 90, C -0, E1 0, E2 0, E3 0, E4 0} C_DIS
LIN {X 767.741, Y -434.323, Z 92, A 0, B 90, C -0, E1 0, E2 0, E3 0, E4 0} C_DIS
LIN {X 769.022, Y -434.515, Z 92, A 0, B 90, C -0, E1 0, E2 0, E3 0, E4 0} C_DIS
LIN {X 775.172, Y -436.825, Z 92, A 0, B 90, C -0, E1 0, E2 0, E3 0, E4 0} C_DIS
LIN {X 776.432, Y -436.86, Z 92, A 0, B 90, C -0, E1 0, E2 0, E3 0, E4 0} C_DIS
LIN {X 776.99, Y -435.707, Z 92, A 0, B 90, C -0, E1 0, E2 0, E3 0, E4 0} C_DIS
LIN {X 778.491, Y -429.311, Z 92, A 0, B 90, C -0, E1 0, E2 0, E3 0, E4 0} C_DIS
LIN {X 779.132, Y -428.19, Z 92, A 0, B 90, C -0, E1 0, E2 0, E3 0, E4 0} C_DIS
LIN {X 780.338, Y -427.715, Z 92, A 0, B 90, C -0, E1 0, E2 0, E3 0, E4 0} C_DIS
LIN {X 786.819, Y -426.641, Z 92, A 0, B 90, C -0, E1 0, E2 0, E3 0, E4 0} C_DIS
LIN {X 787.927, Y -426.042, Z 92, A 0, B 90, C -0, E1 0, E2 0, E3 0, E4 0} C_DIS
LIN {X 787.834, Y -424.764, Z 92, A 0, B 90, C -0, E1 0, E2 0, E3 0, E4 0} C_DIS
LIN {X 785.936, Y -418.474, Z 92, A 0, B 90, C -0, E1 0, E2 0, E3 0, E4 0} C_DIS
LIN {X 785.931, Y -417.183, Z 92, A 0, B 90, C -0, E1 0, E2 0, E3 0, E4 0} C_DIS
LIN {X 786.738, Y -416.169, Z 92, A 0, B 90, C -0, E1 0, E2 0, E3 0, E4 0} C_DIS
LIN {X 791.814, Y -411.998, Z 92, A 0, B 90, C -0, E1 0, E2 0, E3 0, E4 0} C_DIS
LIN {X 792.474, Y -410.925, Z 92, A 0, B 90, C -0, E1 0, E2 0, E3 0, E4 0} C_DIS
LIN {X 791.754, Y -409.866, Z 92, A 0, B 90, C -0, E1 0, E2 0, E3 0, E4 0} C_DIS
LIN {X 786.966, Y -405.367, Z 92, A 0, B 90, C -0, E1 0, E2 0, E3 0, E4 0} C_DIS
LIN {X 786.316, Y -404.251, Z 92, A 0, B 90, C -0, E1 0, E2 0, E3 0, E4 0} C_DIS
LIN {X 786.507, Y -402.97, Z 92, A 0, B 90, C -0, E1 0, E2 0, E3 0, E4 0} C_DIS
LIN {X 788.818, Y -396.82, Z 92, A 0, B 90, C -0, E1 0, E2 0, E3 0, E4 0} C_DIS
LIN {X 788.853, Y -395.561, Z 92, A 0, B 90, C -0, E1 0, E2 0, E3 0, E4 0} C_DIS
LIN {X 787.699, Y -395.003, Z 92, A 0, B 90, C -0, E1 0, E2 0, E3 0, E4 0} C_DIS
LIN {X 781.303, Y -393.501, Z 92, A 0, B 90, C -0, E1 0, E2 0, E3 0, E4 0} C_DIS
LIN {X 780.183, Y -392.86, Z 92, A 0, B 90, C -0, E1 0, E2 0, E3 0, E4 0} C_DIS
LIN {X 779.708, Y -391.655, Z 92, A 0, B 90, C -0, E1 0, E2 0, E3 0, E4 0} C_DIS
LIN {X 778.634, Y -385.173, Z 92, A 0, B 90, C -0, E1 0, E2 0, E3 0, E4 0} C_DIS
LIN {X 778.035, Y -384.065, Z 92, A 0, B 90, C -0, E1 0, E2 0, E3 0, E4 0} C_DIS
LIN {X 776.757, Y -384.159, Z 92, A 0, B 90, C -0, E1 0, E2 0, E3 0, E4 0} C_DIS
LIN {X 771.725, Y -385.677, Z 92, A 0, B 90, C -0, E1 0, E2 0, E3 0, E4 0} C_DIS
LIN {X 770.223, Y -386.109, Z 92.65, A 0, B 90, C -0, E1 0, E2 0, E3 0, E4 0} C_DIS
LIN {X 768.939, Y -386.125, Z 92.65, A 0, B 90, C -0, E1 0, E2 0, E3 0, E4 0} C_DIS
LIN {X 767.923, Y -385.331, Z 92.65, A 0, B 90, C -0, E1 0, E2 0, E3 0, E4 0} C_DIS
LIN {X 763.731, Y -380.316, Z 92.65, A 0, B 90, C -0, E1 0, E2 0, E3 0, E4 0} C_DIS
LIN {X 762.658, Y -379.669, Z 92.65, A 0, B 90, C -0, E1 0, E2 0, E3 0, E4 0} C_DIS
LIN {X 761.61, Y -380.394, Z 92.65, A 0, B 90, C -0, E1 0, E2 0, E3 0, E4 0} C_DIS
LIN {X 757.175, Y -385.195, Z 92.65, A 0, B 90, C -0, E1 0, E2 0, E3 0, E4 0} C_DIS
LIN {X 756.07, Y -385.851, Z 92.65, A 0, B 90, C -0, E1 0, E2 0, E3 0, E4 0} C_DIS
LIN {X 754.794, Y -385.671, Z 92.65, A 0, B 90, C -0, E1 0, E2 0, E3 0, E4 0} C_DIS
LIN {X 748.656, Y -383.424, Z 92.65, A 0, B 90, C -0, E1 0, E2 0, E3 0, E4 0} C_DIS
LIN {X 747.404, Y -383.399, Z 92.65, A 0, B 90, C -0, E1 0, E2 0, E3 0, E4 0} C_DIS
LIN {X 746.858, Y -384.551, Z 92.65, A 0, B 90, C -0, E1 0, E2 0, E3 0, E4 0} C_DIS
LIN {X 745.418, Y -390.927, Z 92.65, A 0, B 90, C -0, E1 0, E2 0, E3 0, E4 0} C_DIS
LIN {X 744.789, Y -392.047, Z 92.65, A 0, B 90, C -0, E1 0, E2 0, E3 0, E4 0} C_DIS
LIN {X 743.594, Y -392.53, Z 92.65, A 0, B 90, C -0, E1 0, E2 0, E3 0, E4 0} C_DIS
LIN {X 737.155, Y -393.652, Z 92.65, A 0, B 90, C -0, E1 0, E2 0, E3 0, E4 0} C_DIS
LIN {X 736.058, Y -394.258, Z 92.65, A 0, B 90, C -0, E1 0, E2 0, E3 0, E4 0} C_DIS
LIN {X 736.161, Y -395.528, Z 92.65, A 0, B 90, C -0, E1 0, E2 0, E3 0, E4 0} C_DIS
LIN {X 738.102, Y -401.77, Z 92.65, A 0, B 90, C -0, E1 0, E2 0, E3 0, E4 0} C_DIS
LIN {X 738.117, Y -403.054, Z 92.65, A 0, B 90, C -0, E1 0, E2 0, E3 0, E4 0} C_DIS
LIN {X 737.324, Y -404.07, Z 92.65, A 0, B 90, C -0, E1 0, E2 0, E3 0, E4 0} C_DIS
LIN {X 732.309, Y -408.261, Z 92.65, A 0, B 90, C -0, E1 0, E2 0, E3 0, E4 0} C_DIS
LIN {X 731.661, Y -409.334, Z 92.65, A 0, B 90, C -0, E1 0, E2 0, E3 0, E4 0} C_DIS
LIN {X 732.386, Y -410.382, Z 92.65, A 0, B 90, C -0, E1 0, E2 0, E3 0, E4 0} C_DIS
LIN {X 737.187, Y -414.818, Z 92.65, A 0, B 90, C -0, E1 0, E2 0, E3 0, E4 0} C_DIS
LIN {X 737.843, Y -415.922, Z 92.65, A 0, B 90, C -0, E1 0, E2 0, E3 0, E4 0} C_DIS
LIN {X 737.664, Y -417.198, Z 92.65, A 0, B 90, C -0, E1 0, E2 0, E3 0, E4 0} C_DIS
LIN {X 735.416, Y -423.336, Z 92.65, A 0, B 90, C -0, E1 0, E2 0, E3 0, E4 0} C_DIS
LIN {X 735.392, Y -424.589, Z 92.65, A 0, B 90, C -0, E1 0, E2 0, E3 0, E4 0} C_DIS
LIN {X 736.544, Y -425.134, Z 92.65, A 0, B 90, C -0, E1 0, E2 0, E3 0, E4 0} C_DIS
LIN {X 742.919, Y -426.575, Z 92.65, A 0, B 90, C -0, E1 0, E2 0, E3 0, E4 0} C_DIS
LIN {X 744.04, Y -427.203, Z 92.65, A 0, B 90, C -0, E1 0, E2 0, E3 0, E4 0} C_DIS
LIN {X 744.522, Y -428.399, Z 92.65, A 0, B 90, C -0, E1 0, E2 0, E3 0, E4 0} C_DIS
LIN {X 745.645, Y -434.838, Z 92.65, A 0, B 90, C -0, E1 0, E2 0, E3 0, E4 0} C_DIS
LIN {X 746.25, Y -435.935, Z 92.65, A 0, B 90, C -0, E1 0, E2 0, E3 0, E4 0} C_DIS
LIN {X 747.521, Y -435.831, Z 92.65, A 0, B 90, C -0, E1 0, E2 0, E3 0, E4 0} C_DIS
LIN {X 753.762, Y -433.891, Z 92.65, A 0, B 90, C -0, E1 0, E2 0, E3 0, E4 0} C_DIS
LIN {X 755.046, Y -433.875, Z 92.65, A 0, B 90, C -0, E1 0, E2 0, E3 0, E4 0} C_DIS
LIN {X 756.062, Y -434.669, Z 92.65, A 0, B 90, C -0, E1 0, E2 0, E3 0, E4 0} C_DIS
LIN {X 760.254, Y -439.684, Z 92.65, A 0, B 90, C -0, E1 0, E2 0, E3 0, E4 0} C_DIS
LIN {X 761.327, Y -440.331, Z 92.65, A 0, B 90, C -0, E1 0, E2 0, E3 0, E4 0} C_DIS
LIN {X 762.375, Y -439.606, Z 92.65, A 0, B 90, C -0, E1 0, E2 0, E3 0, E4 0} C_DIS
LIN {X 766.81, Y -434.805, Z 92.65, A 0, B 90, C -0, E1 0, E2 0, E3 0, E4 0} C_DIS
LIN {X 767.915, Y -434.149, Z 92.65, A 0, B 90, C -0, E1 0, E2 0, E3 0, E4 0} C_DIS
LIN {X 769.191, Y -434.329, Z 92.65, A 0, B 90, C -0, E1 0, E2 0, E3 0, E4 0} C_DIS
LIN {X 775.328, Y -436.576, Z 92.65, A 0, B 90, C -0, E1 0, E2 0, E3 0, E4 0} C_DIS
LIN {X 776.581, Y -436.601, Z 92.65, A 0, B 90, C -0, E1 0, E2 0, E3 0, E4 0} C_DIS
LIN {X 777.127, Y -435.449, Z 92.65, A 0, B 90, C -0, E1 0, E2 0, E3 0, E4 0} C_DIS
LIN {X 778.567, Y -429.073, Z 92.65, A 0, B 90, C -0, E1 0, E2 0, E3 0, E4 0} C_DIS
LIN {X 779.196, Y -427.953, Z 92.65, A 0, B 90, C -0, E1 0, E2 0, E3 0, E4 0} C_DIS
LIN {X 780.391, Y -427.47, Z 92.65, A 0, B 90, C -0, E1 0, E2 0, E3 0, E4 0} C_DIS
LIN {X 786.83, Y -426.348, Z 92.65, A 0, B 90, C -0, E1 0, E2 0, E3 0, E4 0} C_DIS
LIN {X 787.927, Y -425.742, Z 92.65, A 0, B 90, C -0, E1 0, E2 0, E3 0, E4 0} C_DIS
LIN {X 787.823, Y -424.472, Z 92.65, A 0, B 90, C -0, E1 0, E2 0, E3 0, E4 0} C_DIS
LIN {X 785.883, Y -418.23, Z 92.65, A 0, B 90, C -0, E1 0, E2 0, E3 0, E4 0} C_DIS
LIN {X 785.867, Y -416.946, Z 92.65, A 0, B 90, C -0, E1 0, E2 0, E3 0, E4 0} C_DIS
LIN {X 786.661, Y -415.93, Z 92.65, A 0, B 90, C -0, E1 0, E2 0, E3 0, E4 0} C_DIS
LIN {X 791.676, Y -411.739, Z 92.65, A 0, B 90, C -0, E1 0, E2 0, E3 0, E4 0} C_DIS
LIN {X 792.324, Y -410.666, Z 92.65, A 0, B 90, C -0, E1 0, E2 0, E3 0, E4 0} C_DIS
LIN {X 791.599, Y -409.618, Z 92.65, A 0, B 90, C -0, E1 0, E2 0, E3 0, E4 0} C_DIS
LIN {X 786.798, Y -405.182, Z 92.65, A 0, B 90, C -0, E1 0, E2 0, E3 0, E4 0} C_DIS
LIN {X 786.142, Y -404.078, Z 92.65, A 0, B 90, C -0, E1 0, E2 0, E3 0, E4 0} C_DIS
LIN {X 786.321, Y -402.802, Z 92.65, A 0, B 90, C -0, E1 0, E2 0, E3 0, E4 0} C_DIS
LIN {X 788.569, Y -396.664, Z 92.65, A 0, B 90, C -0, E1 0, E2 0, E3 0, E4 0} C_DIS
LIN {X 788.593, Y -395.411, Z 92.65, A 0, B 90, C -0, E1 0, E2 0, E3 0, E4 0} C_DIS
LIN {X 787.441, Y -394.866, Z 92.65, A 0, B 90, C -0, E1 0, E2 0, E3 0, E4 0} C_DIS
LIN {X 781.066, Y -393.425, Z 92.65, A 0, B 90, C -0, E1 0, E2 0, E3 0, E4 0} C_DIS
LIN {X 779.945, Y -392.797, Z 92.65, A 0, B 90, C -0, E1 0, E2 0, E3 0, E4 0} C_DIS
LIN {X 779.463, Y -391.601, Z 92.65, A 0, B 90, C -0, E1 0, E2 0, E3 0, E4 0} C_DIS
LIN {X 778.34, Y -385.162, Z 92.65, A 0, B 90, C -0, E1 0, E2 0, E3 0, E4 0} C_DIS
LIN {X 777.735, Y -384.065, Z 92.65, A 0, B 90, C -0, E1 0, E2 0, E3 0, E4 0} C_DIS
LIN {X 776.464, Y -384.169, Z 92.65, A 0, B 90, C -0, E1 0, E2 0, E3 0, E4 0} C_DIS
LIN {X 771.471, Y -385.721, Z 92.65, A 0, B 90, C -0, E1 0, E2 0, E3 0, E4 0} C_DIS
LIN {X 769.982, Y -386.163, Z 93.3, A 0, B 90, C -0, E1 0, E2 0, E3 0, E4 0} C_DIS
LIN {X 768.704, Y -386.189, Z 93.3, A 0, B 90, C -0, E1 0, E2 0, E3 0, E4 0} C_DIS
LIN {X 767.687, Y -385.408, Z 93.3, A 0, B 90, C -0, E1 0, E2 0, E3 0, E4 0} C_DIS
LIN {X 763.475, Y -380.454, Z 93.3, A 0, B 90, C -0, E1 0, E2 0, E3 0, E4 0} C_DIS
LIN {X 762.402, Y -379.819, Z 93.3, A 0, B 90, C -0, E1 0, E2 0, E3 0, E4 0} C_DIS
LIN {X 761.365, Y -380.549, Z 93.3, A 0, B 90, C -0, E1 0, E2 0, E3 0, E4 0} C_DIS
LIN {X 756.993, Y -385.362, Z 93.3, A 0, B 90, C -0, E1 0, E2 0, E3 0, E4 0} C_DIS
LIN {X 755.9, Y -386.024, Z 93.3, A 0, B 90, C -0, E1 0, E2 0, E3 0, E4 0} C_DIS
LIN {X 754.628, Y -385.856, Z 93.3, A 0, B 90, C -0, E1 0, E2 0, E3 0, E4 0} C_DIS
LIN {X 748.503, Y -383.671, Z 93.3, A 0, B 90, C -0, E1 0, E2 0, E3 0, E4 0} C_DIS
LIN {X 747.257, Y -383.657, Z 93.3, A 0, B 90, C -0, E1 0, E2 0, E3 0, E4 0} C_DIS
LIN {X 746.724, Y -384.808, Z 93.3, A 0, B 90, C -0, E1 0, E2 0, E3 0, E4 0} C_DIS
LIN {X 745.344, Y -391.163, Z 93.3, A 0, B 90, C -0, E1 0, E2 0, E3 0, E4 0} C_DIS
LIN {X 744.728, Y -392.282, Z 93.3, A 0, B 90, C -0, E1 0, E2 0, E3 0, E4 0} C_DIS
LIN {X 743.543, Y -392.772, Z 93.3, A 0, B 90, C -0, E1 0, E2 0, E3 0, E4 0} C_DIS
LIN {X 737.146, Y -393.943, Z 93.3, A 0, B 90, C -0, E1 0, E2 0, E3 0, E4 0} C_DIS
LIN {X 736.06, Y -394.554, Z 93.3, A 0, B 90, C -0, E1 0, E2 0, E3 0, E4 0} C_DIS
LIN {X 736.173, Y -395.817, Z 93.3, A 0, B 90, C -0, E1 0, E2 0, E3 0, E4 0} C_DIS
LIN {X 738.156, Y -402.011, Z 93.3, A 0, B 90, C -0, E1 0, E2 0, E3 0, E4 0} C_DIS
LIN {X 738.182, Y -403.288, Z 93.3, A 0, B 90, C -0, E1 0, E2 0, E3 0, E4 0} C_DIS
LIN {X 737.401, Y -404.305, Z 93.3, A 0, B 90, C -0, E1 0, E2 0, E3 0, E4 0} C_DIS
LIN {X 732.446, Y -408.517, Z 93.3, A 0, B 90, C -0, E1 0, E2 0, E3 0, E4 0} C_DIS
LIN {X 731.811, Y -409.59, Z 93.3, A 0, B 90, C -0, E1 0, E2 0, E3 0, E4 0} C_DIS
LIN {X 732.541, Y -410.627, Z 93.3, A 0, B 90, C -0, E1 0, E2 0, E3 0, E4 0} C_DIS
LIN {X 737.355, Y -415, Z 93.3, A 0, B 90, C -0, E1 0, E2 0, E3 0, E4 0} C_DIS
LIN {X 738.016, Y -416.093, Z 93.3, A 0, B 90, C -0, E1 0, E2 0, E3 0, E4 0} C_DIS
LIN {X 737.848, Y -417.364, Z 93.3, A 0, B 90, C -0, E1 0, E2 0, E3 0, E4 0} C_DIS
LIN {X 735.663, Y -423.489, Z 93.3, A 0, B 90, C -0, E1 0, E2 0, E3 0, E4 0} C_DIS
LIN {X 735.65, Y -424.736, Z 93.3, A 0, B 90, C -0, E1 0, E2 0, E3 0, E4 0} C_DIS
LIN {X 736.8, Y -425.269, Z 93.3, A 0, B 90, C -0, E1 0, E2 0, E3 0, E4 0} C_DIS
LIN {X 743.155, Y -426.649, Z 93.3, A 0, B 90, C -0, E1 0, E2 0, E3 0, E4 0} C_DIS
LIN {X 744.275, Y -427.265, Z 93.3, A 0, B 90, C -0, E1 0, E2 0, E3 0, E4 0} C_DIS
LIN {X 744.765, Y -428.45, Z 93.3, A 0, B 90, C -0, E1 0, E2 0, E3 0, E4 0} C_DIS
LIN {X 745.935, Y -434.846, Z 93.3, A 0, B 90, C -0, E1 0, E2 0, E3 0, E4 0} C_DIS
LIN {X 746.547, Y -435.933, Z 93.3, A 0, B 90, C -0, E1 0, E2 0, E3 0, E4 0} C_DIS
LIN {X 747.81, Y -435.819, Z 93.3, A 0, B 90, C -0, E1 0, E2 0, E3 0, E4 0} C_DIS
LIN {X 754.003, Y -433.837, Z 93.3, A 0, B 90, C -0, E1 0, E2 0, E3 0, E4 0} C_DIS
LIN {X 755.281, Y -433.811, Z 93.3, A 0, B 90, C -0, E1 0, E2 0, E3 0, E4 0} C_DIS
LIN {X 756.298, Y -434.592, Z 93.3, A 0, B 90, C -0, E1 0, E2 0, E3 0, E4 0} C_DIS
LIN {X 760.51, Y -439.546, Z 93.3, A 0, B 90, C -0, E1 0, E2 0, E3 0, E4 0} C_DIS
LIN {X 761.583, Y -440.181, Z 93.3, A 0, B 90, C -0, E1 0, E2 0, E3 0, E4 0} C_DIS
LIN {X 762.62, Y -439.451, Z 93.3, A 0, B 90, C -0, E1 0, E2 0, E3 0, E4 0} C_DIS
LIN {X 766.992, Y -434.638, Z 93.3, A 0, B 90, C -0, E1 0, E2 0, E3 0, E4 0} C_DIS
LIN {X 768.085, Y -433.976, Z 93.3, A 0, B 90, C -0, E1 0, E2 0, E3 0, E4 0} C_DIS
LIN {X 769.357, Y -434.144, Z 93.3, A 0, B 90, C -0, E1 0, E2 0, E3 0, E4 0} C_DIS
LIN {X 775.482, Y -436.329, Z 93.3, A 0, B 90, C -0, E1 0, E2 0, E3 0, E4 0} C_DIS
LIN {X 776.728, Y -436.343, Z 93.3, A 0, B 90, C -0, E1 0, E2 0, E3 0, E4 0} C_DIS
LIN {X 777.261, Y -435.192, Z 93.3, A 0, B 90, C -0, E1 0, E2 0, E3 0, E4 0} C_DIS
LIN {X 778.641, Y -428.837, Z 93.3, A 0, B 90, C -0, E1 0, E2 0, E3 0, E4 0} C_DIS
LIN {X 779.257, Y -427.718, Z 93.3, A 0, B 90, C -0, E1 0, E2 0, E3 0, E4 0} C_DIS
LIN {X 780.442, Y -427.228, Z 93.3, A 0, B 90, C -0, E1 0, E2 0, E3 0, E4 0} C_DIS
LIN {X 786.839, Y -426.057, Z 93.3, A 0, B 90, C -0, E1 0, E2 0, E3 0, E4 0} C_DIS
LIN {X 787.925, Y -425.446, Z 93.3, A 0, B 90, C -0, E1 0, E2 0, E3 0, E4 0} C_DIS
LIN {X 787.812, Y -424.183, Z 93.3, A 0, B 90, C -0, E1 0, E2 0, E3 0, E4 0} C_DIS
LIN {X 785.829, Y -417.989, Z 93.3, A 0, B 90, C -0, E1 0, E2 0, E3 0, E4 0} C_DIS
LIN {X 785.803, Y -416.712, Z 93.3, A 0, B 90, C -0, E1 0, E2 0, E3 0, E4 0} C_DIS
LIN {X 786.584, Y -415.695, Z 93.3, A 0, B 90, C -0, E1 0, E2 0, E3 0, E4 0} C_DIS
LIN {X 791.539, Y -411.483, Z 93.3, A 0, B 90, C -0, E1 0, E2 0, E3 0, E4 0} C_DIS
LIN {X 792.174, Y -410.41, Z 93.3, A 0, B 90, C -0, E1 0, E2 0, E3 0, E4 0} C_DIS
LIN {X 791.444, Y -409.373, Z 93.3, A 0, B 90, C -0, E1 0, E2 0, E3 0, E4 0} C_DIS
LIN {X 786.63, Y -405, Z 93.3, A 0, B 90, C -0, E1 0, E2 0, E3 0, E4 0} C_DIS
LIN {X 785.969, Y -403.907, Z 93.3, A 0, B 90, C -0, E1 0, E2 0, E3 0, E4 0} C_DIS
LIN {X 786.137, Y -402.636, Z 93.3, A 0, B 90, C -0, E1 0, E2 0, E3 0, E4 0} C_DIS
LIN {X 788.322, Y -396.511, Z 93.3, A 0, B 90, C -0, E1 0, E2 0, E3 0, E4 0} C_DIS
LIN {X 788.335, Y -395.264, Z 93.3, A 0, B 90, C -0, E1 0, E2 0, E3 0, E4 0} C_DIS
LIN {X 787.185, Y -394.731, Z 93.3, A 0, B 90, C -0, E1 0, E2 0, E3 0, E4 0} C_DIS
LIN {X 780.83, Y -393.351, Z 93.3, A 0, B 90, C -0, E1 0, E2 0, E3 0, E4 0} C_DIS
LIN {X 779.71, Y -392.735, Z 93.3, A 0, B 90, C -0, E1 0, E2 0, E3 0, E4 0} C_DIS
LIN {X 779.22, Y -391.55, Z 93.3, A 0, B 90, C -0, E1 0, E2 0, E3 0, E4 0} C_DIS
LIN {X 778.05, Y -385.154, Z 93.3, A 0, B 90, C -0, E1 0, E2 0, E3 0, E4 0} C_DIS
LIN {X 777.438, Y -384.067, Z 93.3, A 0, B 90, C -0, E1 0, E2 0, E3 0, E4 0} C_DIS
LIN {X 776.175, Y -384.181, Z 93.3, A 0, B 90, C -0, E1 0, E2 0, E3 0, E4 0} C_DIS
LIN {X 771.22, Y -385.767, Z 93.3, A 0, B 90, C -0, E1 0, E2 0, E3 0, E4 0} C_DIS
LIN {X 769.743, Y -386.218, Z 93.95, A 0, B 90, C -0, E1 0, E2 0, E3 0, E4 0} C_DIS
LIN {X 768.472, Y -386.255, Z 93.95, A 0, B 90, C -0, E1 0, E2 0, E3 0, E4 0} C_DIS
LIN {X 767.454, Y -385.486, Z 93.95, A 0, B 90, C -0, E1 0, E2 0, E3 0, E4 0} C_DIS
LIN {X 763.222, Y -380.591, Z 93.95, A 0, B 90, C -0, E1 0, E2 0, E3 0, E4 0} C_DIS
LIN {X 762.15, Y -379.968, Z 93.95, A 0, B 90, C -0, E1 0, E2 0, E3 0, E4 0} C_DIS
LIN {X 761.124, Y -380.703, Z 93.95, A 0, B 90, C -0, E1 0, E2 0, E3 0, E4 0} C_DIS
LIN {X 756.814, Y -385.529, Z 93.95, A 0, B 90, C -0, E1 0, E2 0, E3 0, E4 0} C_DIS
LIN {X 755.731, Y -386.196, Z 93.95, A 0, B 90, C -0, E1 0, E2 0, E3 0, E4 0} C_DIS
LIN {X 754.465, Y -386.039, Z 93.95, A 0, B 90, C -0, E1 0, E2 0, E3 0, E4 0} C_DIS
LIN {X 748.353, Y -383.917, Z 93.95, A 0, B 90, C -0, E1 0, E2 0, E3 0, E4 0} C_DIS
LIN {X 747.113, Y -383.913, Z 93.95, A 0, B 90, C -0, E1 0, E2 0, E3 0, E4 0} C_DIS
LIN {X 746.592, Y -385.063, Z 93.95, A 0, B 90, C -0, E1 0, E2 0, E3 0, E4 0} C_DIS
LIN {X 745.272, Y -391.397, Z 93.95, A 0, B 90, C -0, E1 0, E2 0, E3 0, E4 0} C_DIS
LIN {X 744.668, Y -392.516, Z 93.95, A 0, B 90, C -0, E1 0, E2 0, E3 0, E4 0} C_DIS
LIN {X 743.493, Y -393.013, Z 93.95, A 0, B 90, C -0, E1 0, E2 0, E3 0, E4 0} C_DIS
LIN {X 737.139, Y -394.231, Z 93.95, A 0, B 90, C -0, E1 0, E2 0, E3 0, E4 0} C_DIS
LIN {X 736.063, Y -394.848, Z 93.95, A 0, B 90, C -0, E1 0, E2 0, E3 0, E4 0} C_DIS
LIN {X 736.187, Y -396.104, Z 93.95, A 0, B 90, C -0, E1 0, E2 0, E3 0, E4 0} C_DIS
LIN {X 738.21, Y -402.249, Z 93.95, A 0, B 90, C -0, E1 0, E2 0, E3 0, E4 0} C_DIS
LIN {X 738.247, Y -403.52, Z 93.95, A 0, B 90, C -0, E1 0, E2 0, E3 0, E4 0} C_DIS
LIN {X 737.478, Y -404.539, Z 93.95, A 0, B 90, C -0, E1 0, E2 0, E3 0, E4 0} C_DIS
LIN {X 732.584, Y -408.77, Z 93.95, A 0, B 90, C -0, E1 0, E2 0, E3 0, E4 0} C_DIS
LIN {X 731.961, Y -409.843, Z 93.95, A 0, B 90, C -0, E1 0, E2 0, E3 0, E4 0} C_DIS
LIN {X 732.696, Y -410.869, Z 93.95, A 0, B 90, C -0, E1 0, E2 0, E3 0, E4 0} C_DIS
LIN {X 737.521, Y -415.179, Z 93.95, A 0, B 90, C -0, E1 0, E2 0, E3 0, E4 0} C_DIS
LIN {X 738.188, Y -416.261, Z 93.95, A 0, B 90, C -0, E1 0, E2 0, E3 0, E4 0} C_DIS
LIN {X 738.032, Y -417.527, Z 93.95, A 0, B 90, C -0, E1 0, E2 0, E3 0, E4 0} C_DIS
LIN {X 735.909, Y -423.639, Z 93.95, A 0, B 90, C -0, E1 0, E2 0, E3 0, E4 0} C_DIS
LIN {X 735.906, Y -424.88, Z 93.95, A 0, B 90, C -0, E1 0, E2 0, E3 0, E4 0} C_DIS
LIN {X 737.055, Y -425.401, Z 93.95, A 0, B 90, C -0, E1 0, E2 0, E3 0, E4 0} C_DIS
LIN {X 743.389, Y -426.721, Z 93.95, A 0, B 90, C -0, E1 0, E2 0, E3 0, E4 0} C_DIS
LIN {X 744.508, Y -427.324, Z 93.95, A 0, B 90, C -0, E1 0, E2 0, E3 0, E4 0} C_DIS
LIN {X 745.006, Y -428.499, Z 93.95, A 0, B 90, C -0, E1 0, E2 0, E3 0, E4 0} C_DIS
LIN {X 746.223, Y -434.854, Z 93.95, A 0, B 90, C -0, E1 0, E2 0, E3 0, E4 0} C_DIS
LIN {X 746.841, Y -435.93, Z 93.95, A 0, B 90, C -0, E1 0, E2 0, E3 0, E4 0} C_DIS
LIN {X 748.096, Y -435.806, Z 93.95, A 0, B 90, C -0, E1 0, E2 0, E3 0, E4 0} C_DIS
